	bLedJog : BOOL;
	bLedDistance : BOOL;
	bLedReset : BOOL;
	bLedAlt : BOOL;
	 
	bLedUp : BOOL;
	bLedDown : BOOL;
	bLedLeft : BOOL;
	bLedRight : BOOL;
END_STRUCT
END_TYPE

// ---- POUs/HMI/Provider/HwHmi/Structures/HMI_PROVIDER_HW_IN.TcDUT
TYPE HMI_PROVIDER_HW_IN EXTENDS ST_HMI_IN :
STRUCT
	// HW specific IN
	stP10A_Pult	AT%I* : ST_P10A_Pult_IN;
	
	stP50A_Haupt AT%I* : ST_P50A_Haupt_IN;
	
	stP51A_S1HandBs	AT%I* : ST_P51A_EuchnerHandB_IN;

END_STRUCT
END_TYPE

// ---- POUs/HMI/Provider/HwHmi/Structures/HMI_PROVIDER_HW_OUT.TcDUT
TYPE HMI_PROVIDER_HW_OUT EXTENDS ST_HMI_OUT :
STRUCT
	// HW specific OUT
	stP10A_Pult	AT%Q* : ST_P10A_Pult_OUT;
	
	stP50A_Haupt AT%Q* : ST_P50A_Haupt_OUT;
	
	stP51A_S1HandBs	AT%Q* : ST_P51A_EuchnerHandB_OUT;
	
END_STRUCT
END_TYPE

// ---- POUs/HMI/Provider/HwHmi/Structures/HMI_PROVIDER_HW_IO.TcDUT
TYPE HMI_PROVIDER_HW_IO :
STRUCT
	stIn	: HMI_PROVIDER_HW_IN;
	stOut	: HMI_PROVIDER_HW_OUT;
END_STRUCT
END_TYPE

// ---- POUs/HMI/Provider/HwHmi/Structures/_Base/ST_PxAB_SxHandAsBs_IN.TcDUT
TYPE ST_PxAB_SxHandAsBs_IN :
STRUCT
	//bEs			: BOOL; // Handbediengerät Sx AS/BS - ES
	//bConfirm		: BOOL; // Zustimmung
	//bS4			: BOOL; // res
	//bS5			: BOOL; // res
	bAngleP			: BOOL; // Winkelverstellung Auf; Taste 6
	//bS7			: BOOL; // res
	//bS8			: BOOL; // res
	bAngleN			: BOOL; // Winkelverstellung Ab; Taste 9
	bStpZust01		: BOOL; // Zustellung Schrittweite 0,1mm; Taste 10
	bStpZust001		: BOOL; // Zustellung Schrittweite 0,01mm; Taste 11
	bStpZust0001	: BOOL; // Zustellung Schrittweite 0,001mm; Taste 12
	bZustP			: BOOL; // Zustellung +; Taste 13
	bTravL			: BOOL; // Traversierung links; Taste 14
	
	bResetError		: BOOL; // reset error
	
	bTravR			: BOOL; // Traversierung rechts; Taste 16
	bZustN			: BOOL; // Zustellung -; Taste 17
END_STRUCT
END_TYPE

// ---- POUs/HMI/Provider/HwHmi/Structures/_Base/ST_PxAB_SxHandAsBs_OUT.TcDUT
TYPE ST_PxAB_SxHandAsBs_OUT :
STRUCT
	bLedS4	: BOOL; // LED zu Taste Sx
	bLedS5	: BOOL;
	bLedS6	: BOOL;
	bLedS7	: BOOL;
	bLedS8	: BOOL;
	bLedS9	: BOOL;
	bLedS10	: BOOL;
	bLedS11	: BOOL;
	bLedS12	: BOOL;
	bLedS13	: BOOL;
	bLedS14	: BOOL;
	bLedS15	: BOOL;
	bLedS16	: BOOL;
	bLedS17	: BOOL;
END_STRUCT
END_TYPE

// ---- POUs/HMI/Provider/Tc3Hmi/Structures/Stations/ST_StationToTc3Hmi.TcDUT
TYPE ST_StationToTc3Hmi :
STRUCT
	stStationName			: ST_Text;	//example -> station 001
	
	//astButton				: ARRAY[0..CONST.iMaxIdxLocalButton] OF ST_HMI_BUTTON_OUT; //programmer defined buttons
	
	//stCounter				: ARRAY[0..CONST.iMaxIdxCounter] OF ST_Counter_Item_String;
	//stEingabeStatusColor	: ST_HMI_COLOR_STRING;
	//stEingabeStatus			: ST_Text;
	
END_STRUCT
END_TYPE

// ---- POUs/HMI/Provider/Tc3Hmi/Structures/Stations/ST_StationFromTc3Hmi.TcDUT
TYPE ST_StationFromTc3Hmi :
STRUCT
	astButton						: ARRAY[0..iMaxIdxLocalButton] OF ST_HMI_BUTTON_IN; // station specific buttons
END_STRUCT
END_TYPE

// ---- POUs/HMI/Provider/Tc3Hmi/Structures/ST_FromTc3Hmi.TcDUT
TYPE ST_FromTc3Hmi EXTENDS ST_HMI_IN :
STRUCT
	// general
	eLanguage					: E_Language := E_Language.DE;
	sCurrentPage				: WSTRING;
	sSetTargetPageConfirm		: WSTRING;
	stPopup						: ST_PopUp_FromHmi;
	//stButton_CloseHmi			: ST_Button_FromHmi; //button close hmi
	stControlCounter			: ST_CounterControlIn;	
	
	// stations custom
	//astStation					: ARRAY[0..E_Station.eStation_nMaxIdx] OF ST_StationFromTc3Hmi;
END_STRUCT
END_TYPE

// ---- POUs/HMI/Provider/Tc3Hmi/Structures/ST_Header.TcDUT
TYPE ST_Header :
STRUCT
	stButtonNavUser		: ST_HMI_BUTTON_OUT;
	stMessageBox1		: ST_Text;
	stMessageBox1Color	: ST_HMI_COLOR_STRING;
	stMessageBox2		: ST_Text;
	stMessageBox2Color	: ST_HMI_COLOR_STRING;
	stMessageBox3		: ST_Text;
	stMessageBox3Color	: ST_HMI_COLOR_STRING;
	stStationName		: ST_Text;
	sDateAndTime		: STRING;
	nLanguageList		: INT; //count of laguages
	aLanguageList		: ARRAY[0..5] OF ST_Text;
END_STRUCT
END_TYPE

// ---- POUs/HMI/Provider/Tc3Hmi/Structures/ST_HMI_Tc3.TcDUT
TYPE ST_HMI_Tc3 :
STRUCT
	stIn	: ST_FromTc3Hmi;
	stOut	: ST_ToTc3Hmi;
END_STRUCT
END_TYPE

// ---- POUs/HMI/Provider/Tc3Hmi/Structures/ST_ToTc3Hmi.TcDUT
TYPE ST_ToTc3Hmi EXTENDS ST_HMI_OUT:
STRUCT
	sSetTargetPage				: WSTRING := "Pages/Stations/conStationOverview.content";
	stHeader					: ST_Header;
	
	stPopup						: ST_PopUp_ToHmi;
	
	stCounter					: ARRAY[0..CONST.iMaxIdxCounter] OF ST_Counter_Item_String;
	stControlCounter			: ST_CounterControlOut;
	
	stConditionMonitoring		: ST_ToTc3HmiConditionMonitoring;
	stSetupPlant				: ARRAY[0..30] OF ST_SetupPlant_Item_String;
	stEmergencyStop				: ARRAY[0..20] OF ST_ToTc3Hmi_EmergencyStop;
	stDoor						: ARRAY[0..20] OF ST_ToTc3Hmi_Door;
	
	//stations
	//astStation					: ARRAY[0..E_Station.eStation_nMaxIdx] OF ST_StationToTc3Hmi;
END_STRUCT
END_TYPE

// ---- POUs/HMI/Provider/Tc3Hmi/Structures/ST_ToTc3HmiConditionMonitoring.TcDUT
TYPE ST_ToTc3HmiConditionMonitoring :
STRUCT
	fVoltage_L1	:REAL;
	fVoltage_L2	:REAL;
	fVoltage_L3	:REAL;
	fVoltage_L1_L2 :REAL;
	fVoltage_L2_L3 :REAL;
	fVoltage_L3_L1 :REAL;
	fPowerFactor :REAL;
	fCurrent_L1 :REAL;
	fCurrent_L2 :REAL;
	fCurrent_L3 :REAL;
	fRealPower_L1 :REAL;	//Wirkleistung
	fRealPower_L2 :REAL;	//Wirkleistung
	fRealPower_L3 :REAL;	//Wirkleistung
	fIdlePower_L1 :REAL;	//Blindleistung
	fIdlePower_L2 :REAL;	//Blindleistung
	fIdlePower_L3 :REAL;	//Blindleistung
	fApparentPower_L1 :REAL;	//Scheinleistung
	fApparentPower_L2 :REAL;	//Scheinleistung
	fArrarentPower_L3 :REAL;	//Scheinleistung
END_STRUCT
END_TYPE

// ---- POUs/HMI/Provider/Tc3Hmi/Structures/ST_ToTc3Hmi_Door.TcDUT
TYPE ST_ToTc3Hmi_Door :
STRUCT
	stName			: ST_Text;
	stItem			: ST_Text;
	stStateColor	: ST_HMI_COLOR_STRING;
END_STRUCT
END_TYPE

// ---- POUs/HMI/Provider/Tc3Hmi/Structures/ST_ToTc3Hmi_EmergencyStop.TcDUT
TYPE ST_ToTc3Hmi_EmergencyStop :
STRUCT
	stName			: ST_Text;
	stItem			: ST_Text;
	nState			: INT;	
END_STRUCT
END_TYPE

// ---- POUs/HMI/Provider/Tc3Hmi/Structures/UserControls/DataGrid/ST_UserControlGrid_FromHmi.TcDUT
TYPE ST_UserControlGrid_FromHmi :
STRUCT
	stButtonSave	: ST_HMI_BUTTON_IN;
END_STRUCT
END_TYPE

// ---- POUs/HMI/Provider/Tc3Hmi/Structures/UserControls/DataGrid/ST_UserControlGrid_ToHmi.TcDUT
TYPE ST_UserControlGrid_ToHmi :
STRUCT
	stButtonSave	: ST_HMI_BUTTON_OUT;
END_STRUCT
END_TYPE

// ---- POUs/HMI/Provider/Tc3Hmi/Structures/UserControls/ManualControl Axis/ST_UserControl_Manual_Axis_FromHmi.TcDUT
TYPE ST_UserControl_Manual_Axis_FromHmi :
STRUCT
	fTargetPosition				: REAL;
	eJogMode					: E_Axis_JogMode;
	stButtonJogPos,
	stButtonJogNeg,
	stButtonGoTo,
	stButtonGear,
	stButtonBrake,			
	stButtonSetPos,	
	stButtonRefReset			: ST_HMI_BUTTON_IN;
	nSelectedRowIndex			: UINT;
	nSelectedColumnIndex		: UINT;		
	bTargetListClick			: BOOL;
	bSetTargetClick				: BOOL;
END_STRUCT
END_TYPE

// ---- POUs/HMI/Provider/Tc3Hmi/Structures/UserControls/ManualControl Axis/ST_UserControl_Manual_Axis_Item.TcDUT
TYPE ST_UserControl_Manual_Axis_Item :
STRUCT
	stName	: ST_Text;
	fPos	: LREAL;
END_STRUCT
END_TYPE

// ---- POUs/HMI/Provider/Tc3Hmi/Structures/UserControls/ManualControl Axis/ST_UserControl_Manual_Axis_Item_String.TcDUT
TYPE ST_UserControl_Manual_Axis_Item_String :
STRUCT
	stName				: ST_Text;
	stPos				: ST_Text;
END_STRUCT
END_TYPE

// ---- POUs/HMI/Provider/Tc3Hmi/Structures/UserControls/ManualControl Axis/ST_UserControl_Manual_Axis_ToHmi.TcDUT
TYPE ST_UserControl_Manual_Axis_ToHmi :
STRUCT
	bVisible					: BOOL;
	bVisibleGear				: BOOL;
	bVisibleRefReset			: BOOL;
	bVisibleBrake				: BOOL;
	bVisibleSetPos				: BOOL;
	stObjectName,
	stGearStatus				: ST_Text;
	sOverride					: STRING;
	sTargetPosition				: STRING;
	sActPosition				: STRING;
	stButtonJogPos,
	stButtonJogNeg,
	stButtonGoTo,
	stButtonGear,				
	stButtonBrake,
	stButtonSetPos,
	stButtonRefReset			: ST_HMI_BUTTON_OUT;	
	aJogModeName				: ARRAY[0..5] OF ST_Text;
	stRefStatus					: ST_Text;	
	stTargetList				: ARRAY[1..10] OF ST_UserControl_Manual_Axis_Item_String; /// product data
END_STRUCT
END_TYPE

// ---- POUs/HMI/Provider/Tc3Hmi/Structures/UserControls/ManualControl Cylinder/ST_UserControl_Manual_Cylinder_FromHmi.TcDUT
TYPE ST_UserControl_Manual_Cylinder_FromHmi :
STRUCT
	stButton_Hp,
	stButton_Mp,
	stButton_Wp	: ST_HMI_BUTTON_IN;
END_STRUCT
END_TYPE

// ---- POUs/HMI/Provider/Tc3Hmi/Structures/UserControls/ManualControl Cylinder/ST_UserControl_Manual_Cylinder_ToHmi.TcDUT
TYPE ST_UserControl_Manual_Cylinder_ToHmi :
STRUCT
	bVisible : BOOL;
	stObjectName				: ST_Text;
	stButton_Hp,
	stButton_Mp,
	stButton_Wp	: ST_HMI_BUTTON_OUT;
	bVisible_Button_Mp			: bool;
END_STRUCT
END_TYPE

// ---- POUs/HMI/Provider/Tc3Hmi/Structures/UserControls/ManualControl Device/ST_UserControl_Manual_Device_FromHmi.TcDUT
TYPE ST_UserControl_Manual_Device_FromHmi :
STRUCT
	stOn,
	stOff		: ST_HMI_BUTTON_IN;	
END_STRUCT
END_TYPE

// ---- POUs/HMI/Provider/Tc3Hmi/Structures/UserControls/ManualControl Device/ST_UserControl_Manual_Device_ToHmi.TcDUT
TYPE ST_UserControl_Manual_Device_ToHmi :
STRUCT
	bVisible 		: BOOL;
	stObjectName	: ST_Text;
	stState			: ST_Text;
	stOn,
	stOff			: ST_HMI_BUTTON_OUT;	
END_STRUCT
END_TYPE

// ---- POUs/HMI/Provider/Tc3Hmi/Structures/UserControls/ManualControl Drive/ST_UserControl_Manual_Drive_FromHmi.TcDUT
TYPE ST_UserControl_Manual_Drive_FromHmi :
STRUCT
	eJogMode					: E_Drive_JogMode;
	stButton_Tipp_Pos,
	stButton_Tipp_Neg,
	stButton_Stop				: ST_HMI_BUTTON_IN;
END_STRUCT
END_TYPE

// ---- POUs/HMI/Provider/Tc3Hmi/Structures/UserControls/ManualControl Drive/ST_UserControl_Manual_Drive_ToHmi.TcDUT
TYPE ST_UserControl_Manual_Drive_ToHmi :
STRUCT
	bVisible : BOOL;
	stObjectName				: ST_Text;
	stState						: ST_Text;
	stButton_Tipp_Pos,
	stButton_Tipp_Neg,
	stButton_Stop				: ST_HMI_BUTTON_OUT;
	aDriveModeName				: ARRAY[0..1] OF ST_Text;
END_STRUCT
END_TYPE

// ---- POUs/HMI/Provider/Tc3Hmi/Structures/UserControls/SensorActor/ST_ToVisuSensorActor.TcDUT
TYPE ST_ToVisuSensorActor :
STRUCT
	stType			: ST_Text;
	stName			: ST_Text;
	stBMK			: ST_Text;
	stZustand		: ST_Text;
END_STRUCT
END_TYPE

// ---- POUs/HMI/Provider/_Enumerations/E_HMI_CONTROL_REQUEST.TcDUT
{attribute 'qualified_only'}
{attribute 'strict'}
TYPE E_HMI_CONTROL_REQUEST :
(
	Default,
	RecipeMgmtRequest,
	SettingMgmtRequest,
	UserMgmtRequest
);   	
END_TYPE

// ---- POUs/HMI/Provider/_Enumerations/E_HMI_PROVIDER.TcDUT
{attribute 'qualified_only'}
{attribute 'strict'}
TYPE E_HMI_PROVIDER :
(
	eHmiProvider_none,
	eHmiProvider_HW,
	eHmiProvider_TC3HMI,
	
	// keep this last:
	eHmiProvider_nMaxIdx
);
END_TYPE

// ---- POUs/HMI/_Enumerations/E_Axis_JogMode.TcTLEO
{attribute 'qualified_only'}
{attribute 'strict'}
TYPE E_Axis_JogMode :
(
	eJogMode_0 := 0,//Kontinuierliche Bewegung
	//eJogMode_1, 	//Tippweg
	eJogMode_1,		//0,01 Tippen
	eJogMode_2,		//0,1 Tippen
	eJogMode_3,		//1 Tippen
	eJogMode_4,		//10 Tippen
	eJogMode_5		//100 Tippen
);
END_TYPE

// ---- POUs/HMI/_Enumerations/E_DataType.TcTLEO
{attribute 'qualified_only'}
{attribute 'strict'}
TYPE E_DataType :
(
	eDataType_None := 0,
	eDataType_bool,
	eDataType_int,
	eDataType_lreal,
	eDataType_wstring,
	eDataType_time_ms,
	eDataType_time_s,
	eDataType_time_m,
	eDataType_time_h,
	
	eDataType_Max
);
END_TYPE

// ---- POUs/HMI/_Enumerations/E_Drive_JogMode.TcDUT
{attribute 'qualified_only'}
{attribute 'strict'}
TYPE E_Drive_JogMode :
(
	eJogMode_0 := 0,//Kontinuierliche Bewegung
	eJogMode_1 		//Tipp Bewegung
);
END_TYPE

// ---- POUs/HMI/_Enumerations/E_Language.TcDUT
//{attribute 'qualified_only'}
//{attribute 'strict'}
TYPE E_Language :
(
	// english
	EN := 0,
	// german
	DE,
	// bulgarisch
	BG,
	
	/// zero based max language index
	eLanguage_maxIdx
);
END_TYPE

// ---- POUs/HMI/_Enumerations/E_ManualObjectControlMode.TcDUT
TYPE E_ManualObjectControlMode :
(
	eManualObjectControlMode_none := 0,
	eManualObjectControlMode_cylinder := 1,
	eManualObjectControlMode_device := 2,
	eManualObjectControlMode_servo := 3
);
END_TYPE

// ---- POUs/HMI/_Enumerations/E_Popup.TcDUT
{attribute 'qualified_only'}
{attribute 'strict'}
TYPE E_Popup :
(
	ePopupNone := 0,
	ePopupSafetyEs,
	ePopupStempelkissenWechseln,
	ePopup02,
	ePopup03,
	ePopup04,
	ePopupMax
);
END_TYPE

// ---- POUs/HMI/_Enumerations/E_RecipeMode.TcTLEO
//{attribute 'qualified_only'}
//{attribute 'strict'}
TYPE E_RecipeMode :
(
	eRecipeMode_None := 0,
	eRecipeMode_ToFrom,
	
	eRecipeMode_Max
);
END_TYPE

// ---- POUs/HMI/_Enumerations/E_User.TcTLEO
//{attribute 'qualified_only'}
//{attribute 'strict'}
TYPE E_User :
(
	eUser_none := 0,	(*User | none*)
	eUser_1,			(*User | 1*)
	eUser_2,			(*User | 2*)
	eUser_3,			(*User | 3*)
	eUser_4,			(*User | 4*)
	eUser_5,			(*User | 5*)
	eUser_6,			(*User | 6*)
	eUser_7,			(*User | 7*)
	eUser_8,			(*User | 8*)
	eUser_9,			(*User | 9*)
	eUser_10,			(*User | 10*)

	eUser_11,			(*User | 11*)
	eUser_12,			(*User | 12*)
	eUser_13,			(*User | 13*)
	eUser_14,			(*User | 14*)
	eUser_15,			(*User | 15*)
	eUser_16,			(*User | 16*)
	eUser_17,			(*User | 17*)
	eUser_18,			(*User | 18*)
	eUser_19,			(*User | 19*)
	eUser_20,			(*User | 20*)	
(*Maximum*)
	eUser_nMaxIdx
);
END_TYPE

// ---- POUs/HMI/_Enumerations/E_User_Level.TcDUT
//{attribute 'qualified_only'}
//{attribute 'strict'}
{attribute 'to_string'}
{attribute 'to_wstring'}
TYPE E_User_Level :
(
	eUser_Level_none := 0,			(*user level 0 = none 1= Operator 2 = Plant Manager 3 = maintenance 4 = reserve 5= admin*)
	eUser_Level_Operator,			(* 1 = Bediener*)
	eUser_Level_Manager,			(* 2 = Einsteller*)
	eUser_Level_Maintenance,		(* 3 = Instandhalter*)
	eUser_Level_Level4,				(* 4 = Reserve*)
	eUser_Level_Admin,				(* 5 = Administrator *)
	eUser_Level_Programmer,			(* 6 = Programmer *)

(*Maximum*)
	eUser_Level_nMaxIdx
);
END_TYPE

// ---- POUs/HMI/_Structures/Counter/E_CounterReaction.TcTLEO
//{attribute 'qualified_only'}
//{attribute 'strict'}
TYPE E_CounterReaction :
(
	eCounterReaction_None := 0,
	eCounterReaction_Info,
	eCounterReaction_Warning,
	eCounterReaction_Error,
	eCounterReaction_SerialFault_Warning,
	eCounterReaction_SerialFault_Error,
	
	eCounterReaction_Max
);
END_TYPE

// ---- POUs/HMI/_Structures/Counter/ST_CounterControlIn.TcDUT
TYPE ST_CounterControlIn :
STRUCT
	stButtonSave		: ST_HMI_BUTTON_IN;
	stButtonReset		: ST_HMI_BUTTON_IN;	
	nSelectedRowIndex	: UINT;
	nSelectedColumIndex	: UINT;
	nInputBool			: DINT;
	nInputNumber		: DINT;
	wsInputString		: WSTRING;
	eUserLevel			: E_User_Level;	
	eReaction			: E_CounterReaction;	
END_STRUCT
END_TYPE

// ---- POUs/HMI/_Structures/Counter/ST_CounterControlOut.TcDUT
TYPE ST_CounterControlOut :
STRUCT
	stButtonSave		: ST_HMI_BUTTON_OUT;
	stButtonReset		: ST_HMI_BUTTON_OUT;		
	bVisible_UserLevel	: BOOL;
	nUserLevelUsers		: INT; //count of recipe mode list
	aUserLevelUsers		: ARRAY[0..E_User_Level.eUser_Level_nMaxIdx] OF ST_Text;
	bVisible_Reaction	: BOOL;
	nReaction			: INT; //count of recipe mode list
	aReaction			: ARRAY[0..E_CounterReaction.eCounterReaction_Max] OF ST_Text;	
	bVisible_Number		: BOOL;
	bVisible_String		: BOOL;
	bVisibleInfo		: BOOL;
	stInfo				: ST_Text;
END_STRUCT
END_TYPE

// ---- POUs/HMI/_Structures/Counter/ST_Counter_Item_String.TcDUT
TYPE ST_Counter_Item_String :
STRUCT
	stIndex					:ST_Text;
	stGroup					:ST_Text;
	stName					:ST_Text;
	stValueOk				:ST_Text;	
	stValueNok				:ST_Text;
	stValueTotal			:ST_Text;	
	stValueOkLevel1			:ST_Text;
	stReactionOkLevel1		:ST_Text;
	stValueOkLevel2			:ST_Text;
	stReactionOkLevel2		:ST_Text;
	stValueNokLevel1		:ST_Text;
	stReactionNokLevel1		:ST_Text;
	stValueNokLevel2		:ST_Text;
	stReactionNokLevel2		:ST_Text;
	stValueTotalLevel1		:ST_Text;
	stReactionTotalLevel1	:ST_Text;
	stValueTotalLevel2		:ST_Text;
	stReactionTotalLevel2	:ST_Text;		
	stUserLevel				:ST_Text;
	stDataType				:ST_Text;	
END_STRUCT
END_TYPE

// ---- POUs/HMI/_Structures/Data/ST_Data_Item_String.TcDUT
TYPE ST_Data_Item_String :
STRUCT
	stIndex				:ST_Text;
	stGroup				:ST_Text;
	stName				:ST_Text;
	stValue				:ST_Text;
	stValueMin			:ST_Text;
	stValueMax			:ST_Text;	
	stUnit				:ST_Text;
	stUserLevel			:ST_Text;
	stDataType			:ST_Text;
	stRecipeMode		:ST_Text;
END_STRUCT
END_TYPE

// ---- POUs/HMI/_Structures/Monitoring/ST_GridObject_Name_Value1_Event1_Value2_Event2_Unit.TcDUT
TYPE ST_GridObject_Name_Value1_Event1_Value2_Event2_Unit :
STRUCT
	sGroup				:STRING;
	sName				:STRING;
	fValue1				:LREAL;
	fValue1Min			:LREAL;
	fValue1Max			:LREAL;
	iEvent1				:INT;	//exampe : no reaction=0 reaction 1..x = 1..x
	fValue2				:LREAL;
	fValue2Min			:LREAL;
	fValue2Max			:LREAL;
	iEvent2				:INT;	//exampe : no reaction=0 reaction 1..x = 1..x
	bYesNo				:BOOL;
	sUnit				:STRING;
END_STRUCT
END_TYPE

// ---- POUs/HMI/_Structures/Monitoring/ST_GridObject_Name_sValue_Unit.TcDUT
TYPE ST_GridObject_Name_sValue_Unit :
STRUCT
	sGroup				:STRING;
	sName				:STRING;
	sValue				:STRING;
	sValueMin			:STRING;
	sValueMax			:STRING;
	bYesNo				:BOOL;
	sUnit				:STRING;
END_STRUCT
END_TYPE

// ---- POUs/HMI/_Structures/Monitoring/ST_Monitoring_Station.TcDUT
TYPE ST_Monitoring_Station EXTENDS ST_Monitoring_Base :
STRUCT
	astMonitoring		: ARRAY[0..CONST.iMaxIdxMonitoring] OF ST_Data_Item;
	astMonitoringView	: ARRAY[0..CONST.iMaxIdxMonitoring] OF ST_Data_Item_String;
END_STRUCT
END_TYPE

// ---- POUs/HMI/_Structures/Monitoring/ST_Monitoring.TcDUT
TYPE ST_Monitoring :
STRUCT
	astMonitoringGlobal		: ARRAY[0..CONST.iMaxIdxMonitoring] OF ST_Data_Item;				// general/global monitoring
	astMonitoringModule		: ARRAY[0..E_Module.eModule_nMaxIdx] OF ST_Monitoring_Module;		// module monitoring
	astMonitoringStation	: ARRAY[0..E_Station.eStation_nMaxIdx] OF ST_Monitoring_Station;	// station monitoring
END_STRUCT
END_TYPE

// ---- POUs/HMI/_Structures/Data/ST_Data_Item.TcDUT
TYPE ST_Data_Item :
STRUCT
	stIndex		: ST_Text;
	stGroup		: ST_Text;
	stName		: ST_Text;
	
	bValue		: BOOL;
	tValue		: TIME;
	sValue		: WSTRING;
	nValue		: INT;
	fValue		: LREAL;
	fValueMin	: LREAL;
	fValueMax	: LREAL;
	
	stUnit		: ST_Text;
	eUserLevel	: E_User_Level;
	eDataType	: E_DataType;
	eRecipeMode	: E_RecipeMode;
END_STRUCT
END_TYPE

// ---- POUs/HMI/_Structures/Monitoring/ST_Monitoring_Base.TcDUT
TYPE ST_Monitoring_Base :
STRUCT
	sGroup				: STRING;
	stName				: ST_Text;
	bManual				: BOOL;
	bInHome				: BOOL;
	bAuto				: BOOL;;
	bBusy				: BOOL;
	bWarning			: BOOL;
	bError				: BOOL;
	bTransferEnable		: BOOL;
END_STRUCT
END_TYPE

// ---- POUs/HMI/_Structures/Monitoring/ST_Monitoring_Module.TcDUT
TYPE ST_Monitoring_Module EXTENDS ST_Monitoring_Base :
STRUCT
	astMonitoring		: ARRAY[0..CONST.iMaxIdxMonitoring] OF ST_Data_Item;
	astMonitoringView	: ARRAY[0..CONST.iMaxIdxMonitoring] OF ST_Data_Item_String;
END_STRUCT
END_TYPE

// ---- POUs/HMI/_Structures/Popup/E_PopupSymbol.TcDUT
{attribute 'qualified_only'}
{attribute 'strict'}
TYPE E_PopupSymbol :
(
	ePopupSymbolNone := 0,
	ePopupSymbolOk,
	ePopupSymbolNok
);
END_TYPE

// ---- POUs/HMI/_Structures/Popup/ST_PopUp_FromHmi.TcDUT
TYPE ST_PopUp_FromHmi :
STRUCT
	stButton01	: ST_HMI_BUTTON_IN;
	stButton02	: ST_HMI_BUTTON_IN;
	stButton03	: ST_HMI_BUTTON_IN;
	stButton04	: ST_HMI_BUTTON_IN;
END_STRUCT
END_TYPE

// ---- POUs/HMI/_Structures/Popup/ST_PopUp_ToHmi.TcDUT
TYPE ST_PopUp_ToHmi :
STRUCT
	bVisible		: BOOL;
	nSymbol			: INT; //E_PopupSymbol;
	stText			: ST_Text;
	bButton01		: BOOL := TRUE;
	stButton01		: ST_HMI_BUTTON_OUT;
	bButton02		: BOOL := TRUE;
	stButton02		: ST_HMI_BUTTON_OUT;
	bButton03		: BOOL := TRUE;
	stButton03		: ST_HMI_BUTTON_OUT;
	bButton04		: BOOL := TRUE;
	stButton04		: ST_HMI_BUTTON_OUT;
END_STRUCT
END_TYPE

// ---- POUs/HMI/_Structures/Recipe/ST_HMI_RECIPE_IN.TcDUT
TYPE ST_HMI_RECIPE_IN :
STRUCT
	// Current Recipe Infos
	bSaveCurrentRecipe				:BOOL;
	
	
	// Recipe Management
	
	wsNewEditRecipeName				:WSTRING(255); // Read/Write
	wsNewEditRecipeComment			:WSTRING(255); // Read/Write
	wsNewEditRecipeProduct			:WSTRING(255); // Read/Write
	bCreateNewRecipe				:BOOL;
	bUpdateRecipe					:BOOL;
	
	nSelectedRecipe					:INT;
	bRefreshRecipeList				:BOOL;
	bLoadSelectedRecipe				:BOOL;
	bDeleteSelectedRecipe			:BOOL;
	wsCopyRecipeNewName				:WSTRING(255); // Read/Write
	bCopySelectedRecipe				:BOOL;
	
END_STRUCT
END_TYPE

// ---- POUs/HMI/_Structures/Recipe/ST_HMI_RECIPE_OUT.TcDUT
TYPE ST_HMI_RECIPE_OUT :
STRUCT
	// Current Recipe Infos
	
	wsActiveRecipe					: WSTRING(255); // Read/Write
	wsActiveRecipeComment			: WSTRING(255); // Read/Write
	wsActiveRecipeProduct			: WSTRING(255); // Read/Write
	wsActiveRecipeSavedInfo			: WSTRING(80);
	bEnableSaveCurrentRecipe		: BOOL;
	                                  
	                                  
	// Recipe Management              
	bEnableCreateNewRecipe			: BOOL;
	bEnableUpdateRecipe				: BOOL;
                                      
	aRecipeList						: ARRAY[0..iMaxIdxRecipe] OF WSTRING(255);
	nMaxEntryRecipeList				: INT;
	bEnableLoadRecipe				: BOOL;
	bEnableDeleteRecipe				: BOOL;
	bEnableCopyRecipe				: BOOL;
                                      
	stStatusText					: ST_Text;
	stStatusColor					: ST_HMI_COLOR_STRING;
	bStatusTextVisible				: BOOL;
END_STRUCT
END_TYPE

// ---- POUs/HMI/_Structures/Safety/ST_HMI_SAFETY_IN.TcDUT
TYPE ST_HMI_SAFETY_IN :
STRUCT
	bQuitSafety,
	
	bQuitAreaST10,
	bUnlockDoorST33	: BOOL;
END_STRUCT
END_TYPE

// ---- POUs/HMI/_Structures/Safety/ST_HMI_SAFETY_OUT.TcDUT
TYPE ST_HMI_SAFETY_OUT :
STRUCT
	// Safety Infos
	
	/// EmergencyStop/Not-Halt Status von Safety (TRUE = OK)
	bSAFE_ES_Ok				: BOOL;
	
	/// State of every emergency stop button (TRUE = OK)
	bSAFE_EStop_State		: ARRAY[0..E_EmergencyStop.eEmergencyStop_nMaxIdx] OF BOOL;
	
	/// Schutzbereich OK von Safety (TRUE = OK)
	bSAFE_AREA_Ok			: ARRAY[0..iSafety_Anzahl_Schutzbereiche] OF BOOL;
	bSAFE_AREA_Ok_Color		: ARRAY[0..iSafety_Anzahl_Schutzbereiche] OF ST_HMI_COLOR_STRING;
	
	/// GATE OK von Safety (TRUE = OK)
	stSAFE_GATE_Ok_Color	: ARRAY[0..E_Door.eDoor_nMaxIdx] OF ST_HMI_COLOR_STRING;
			
	/// Zustimmeinrichtung von Safety (TRUE = OK)
	bSAFE_CONFIRMDEVICE_OK	: BOOL;
	
	bLedResetSafety,
	bLedResetAreaST10,
	bLedResetAreaST33		: BOOL;
END_STRUCT
END_TYPE

// ---- POUs/HMI/_Structures/Settngs/ST_HMI_CONTROL_SETTING_IN.TcDUT
TYPE ST_HMI_CONTROL_SETTING_IN :
STRUCT
	stControlSetting_Plant		: ST_HMI_CONTROL_SETTING_ITEM_IN;
	stControlSetting_Product	: ST_HMI_CONTROL_SETTING_ITEM_IN;
	stControlSetting_Production	: ST_HMI_CONTROL_SETTING_ITEM_IN;	
	
	astControlSetting_Modules	: ARRAY[0..E_Module.eModule_nMaxIdx] OF ST_HMI_CONTROL_SETTING_ITEM_IN;
	astControlSetting_Stations	: ARRAY[0..E_Station.eStation_nMaxIdx] OF ST_HMI_CONTROL_SETTING_ITEM_IN;
END_STRUCT
END_TYPE

// ---- POUs/HMI/_Structures/Settngs/ST_HMI_CONTROL_SETTING_OUT.TcDUT
TYPE ST_HMI_CONTROL_SETTING_OUT :
STRUCT
	stControlSetting_Plant		: ST_HMI_CONTROL_SETTING_ITEM_OUT;
	stControlSetting_Product	: ST_HMI_CONTROL_SETTING_ITEM_OUT;
	stControlSetting_Production	: ST_HMI_CONTROL_SETTING_ITEM_OUT;

	stSettingViewPlant			: ARRAY[0..E_PlantSettings.ePlantSetting_nMaxIdx] OF ST_Data_Item_String;
	stSettingViewProduct		: ARRAY[0..E_ProductSettings.eProductSettings_nMaxIdx] OF ST_Data_Item_String;
	stSettingViewProduction		: ARRAY[0..E_ProductionSettings.eProductionSettings_nMaxIdx] OF ST_Data_Item_String;	

	astSettingModules			: ARRAY[0..E_Module.eModule_nMaxIdx] OF ST_HMI_CONTROL_SETTING_MODULE_OUT;
	astSettingStations			: ARRAY[0..E_Station.eStation_nMaxIdx] OF ST_HMI_CONTROL_SETTING_STATION_OUT;
END_STRUCT
END_TYPE

// ---- POUs/HMI/_Structures/Settngs/ST_HMI_CONTROL_SETTING_STATION_OUT.TcDUT
TYPE ST_HMI_CONTROL_SETTING_STATION_OUT :
STRUCT
	stControlSetting	: ST_HMI_CONTROL_SETTING_ITEM_OUT;
	stSettingView		: ARRAY[0..CONST.iMaxIdxLocalSetting] OF ST_Data_Item_String;
END_STRUCT
END_TYPE

// ---- POUs/HMI/_Structures/Settngs/ST_HMI_CONTROL_SETTING_MODULE_OUT.TcDUT
TYPE ST_HMI_CONTROL_SETTING_MODULE_OUT :
STRUCT
	stControlSetting	: ST_HMI_CONTROL_SETTING_ITEM_OUT;
	stSettingView		: ARRAY[0..CONST.iMaxIdxLocalSetting] OF ST_Data_Item_String;
END_STRUCT
END_TYPE

// ---- POUs/HMI/_Structures/SetupPlant/E_SetupPlantShape.TcDUT
TYPE E_SetupPlantShape :
(
	eSetupPlantShape_None := 0,
	eSetupPlantShape_DreieckGruen,
	eSetupPlantShape_DreieckRot,
	
	eSetupPlantShape_ViereckViolett := 11,
	eSetupPlantShape_ViereckRosa,
	
	eSetupPlantShape_SechseckBlau := 21,
	eSetupPlantShape_SechseckGelb,	
	
	eSetupPlantShape_KreisGruen := 31,
	eSetupPlantShape_KreisRosa,	
	
	eSetupPlantShape_Max
);
END_TYPE

// ---- POUs/HMI/_Structures/SetupPlant/E_SetupPlantStateShape.TcDUT
TYPE E_SetupPlantStateShape :
(
	eSetupPlantStateShape_None := 0,
	eSetupPlantStateShape_Nok,
	eSetupPlantStateShape_Ok,
	
	
	eSetupPlantStateShape_Max
);
END_TYPE

// ---- POUs/HMI/_Structures/SetupPlant/ST_SetupPlant_Item_String.TcDUT
TYPE ST_SetupPlant_Item_String :
STRUCT
	stGroup					:ST_Text;	
	stStation				:ST_Text;
	stName					:ST_Text;
	stSet					:ST_Text;
	stGet					:ST_Text;	
	stState					:ST_Text;		
	stUserLevel				:ST_Text;
	stDataType				:ST_Text;	
END_STRUCT
END_TYPE

// ---- POUs/HMI/_Structures/Settngs/ST_HMI_CONTROL_SETTING_ITEM_IN.TcDUT
TYPE ST_HMI_CONTROL_SETTING_ITEM_IN :
STRUCT
	stButtonSave		: ST_HMI_BUTTON_IN;
	nSelectedRowIndex	: UINT;
	nSelectedColumIndex	: UINT;
	bInputBool			: BOOL;
	nInputNumber		: INT;
	fInputFloat			: REAL;
	wsInputString		: WSTRING;
	eUserLevel			: E_User_Level;
	eRecipeMode			: E_RecipeMode;
END_STRUCT
END_TYPE

// ---- POUs/HMI/_Structures/Settngs/ST_HMI_CONTROL_SETTING_ITEM_OUT.TcDUT
TYPE ST_HMI_CONTROL_SETTING_ITEM_OUT :
STRUCT
	stButtonSave		: ST_HMI_BUTTON_OUT;
	bVisible_RecipeMode	: BOOL;
	nRecipeMode			: INT; //count of recipe mode list
	aRecipeMode			: ARRAY[0..E_RecipeMode.eRecipeMode_Max] OF ST_Text;
	
	bVisible_UserLevel	: BOOL;
	bVisible_Bool		: BOOL;
	bVisible_Float		: BOOL;
	bVisible_Number		: BOOL;
	bVisible_String		: BOOL;
	bVisibleInfo		: BOOL;
	stInfo				: ST_Text;
	
	nUserLevelUsers		: INT; //count of recipe mode list
	aUserLevelUsers		: ARRAY[0..E_User_Level.eUser_Level_nMaxIdx] OF ST_Text;
END_STRUCT
END_TYPE

// ---- POUs/HMI/_Structures/ST_HMI.TcDUT
TYPE ST_HMI :
STRUCT
	stIn 	: ST_HMI_IN;
	stOut 	: ST_HMI_OUT;
END_STRUCT
END_TYPE

// ---- POUs/HMI/_Structures/ST_HMI_IN.TcDUT
TYPE ST_HMI_IN EXTENDS ST_HMI_BASE_IN :
STRUCT
	// additional, project specific stuff:
	iOverride		: INT;
	
	stM001 	: ST_M001_HMI_IN;
	stSt010 : ST_St010_HMI_IN;
	stSt020 : ST_St020_HMI_IN;
	stSt030 : ST_St030_HMI_IN;
	stSt040 : ST_St040_HMI_IN;
END_STRUCT
END_TYPE

// ---- POUs/HMI/_Structures/ST_HMI_InOut.TcDUT
TYPE ST_HMI_InOut :
STRUCT
	/// HMI direct (IN/OUT) struct
	/// e.g. for accessing (r/w) project specific settings

	//stM001 	: ST_M001_HMI_InOut;
	
	stSt010		: ST_St010_HMI_IN_OUT;
	stSt020		: ST_St020_HMI_IN_OUT;
	stSt030		: ST_St030_HMI_IN_OUT;
	stSt040		: ST_St040_HMI_IN_OUT;
	
	// global axis manager
	stHmiAxisManager	: ST_HmiAxisManager;
END_STRUCT
END_TYPE

// ---- POUs/HMI/_Structures/ST_HMI_OUT.TcDUT
TYPE ST_HMI_OUT : //EXTENDS ST_HMI_BASE_OUT :
STRUCT
	// note, ST_HMI_BASE_OUT is not inherited anymoredue to performance issues in provider mapping
	stCommon			: REFERENCE TO ST_HMI_BASE_OUT;
	
	// additional, project specific stuff:
	stButtonDoorOpen	: ST_HMI_BUTTON_OUT;
	stButtonDoorClose	: ST_HMI_BUTTON_OUT;
	stButtonConfirm		: ST_HMI_BUTTON_OUT;
	
	stM001 : ST_M001_HMI_OUT;
	stSt010 : ST_St010_HMI_OUT;
	stSt020 : ST_St020_HMI_OUT;
	stSt030 : ST_St030_HMI_OUT;
	stSt040 : ST_St040_HMI_OUT;
END_STRUCT
END_TYPE

// ---- POUs/HMI/_Structures/ST_NameValue.TcDUT
TYPE ST_NameValue :
STRUCT
	sName 	: STRING(31);
	sValue 	: STRING; 
END_STRUCT
END_TYPE

// ---- POUs/HMI/_Structures/UserManagment/ST_HMI_USER_MGMT_IN.TcDUT
TYPE ST_HMI_USER_MGMT_IN :
STRUCT
	stControlObject					: ST_HMI_GRID_IN;
	sUserManagment_InputString		: STRING;	//Input String Values
	sUserManagment_InputPassword	: STRING;	//Input Password Login
	nUserManagment_InputNumeric		: INT;		//Input Numeric Values
	nUserManagment_InputUserLevel	: INT;		//Input DropDown UserLevel
	stButton_LogOut					: ST_HMI_BUTTON_IN;		//Logout Button
	stButton_LogIn					: ST_HMI_BUTTON_IN;		//Login Button
	stButton_Submit					: ST_HMI_BUTTON_IN;		//Übernehmen Button

	bDeleteUser						: BOOL;
	sCreateDeleteUserName			: STRING;
	sCreateDeleteUserNameConfirm	: STRING;
	sCreateUser_InputPassword		: STRING;	//Input Password Login for create new user
	
	// for Beckhoff HMI UserMgmt:
	iHmiUserLevel					: INT;
END_STRUCT
END_TYPE

// ---- POUs/HMI/_Structures/UserManagment/ST_HMI_USER_MGMT_OUT.TcDUT
TYPE ST_HMI_USER_MGMT_OUT :
STRUCT
	sUserState						: STRING;
	stButton_LogOut					: ST_HMI_BUTTON_OUT;
	stButton_LogIn					: ST_HMI_BUTTON_OUT;
	stButton_Submit					: ST_HMI_BUTTON_OUT;
	stUserLevel						: ARRAY [0..20] OF ST_User_Management;
	bUserLevel						: ARRAY [0..E_User_Level.eUser_Level_nMaxIdx] OF BOOL;
	aUserLevelList					: ARRAY[0..E_User_Level.eUser_Level_nMaxIdx] OF ST_Text;
	bKeyboardInputVisible			: BOOL;
	bNumpadInputVisible				: BOOL;
	bUserLevelInputVisible			: BOOL;
	bPasswordInputVisible			: BOOL;
	stUserManagementMessage			: ST_Text;
	
	stInputDisplayText				: ST_Text;

	bCreateDeleteUserVisible		: BOOL;
	stInfo							: ST_Text;
END_STRUCT
END_TYPE

// ---- POUs/HMI/_Structures/UserManagment/ST_User_Management.TcDUT
{attribute 'pack_mode' := '1'}
TYPE ST_User_Management :
STRUCT
	sName 				: STRING;
	sPassword			: STRING;
	iUserLevel			: E_User_Level;
	stUserLevelName		: ST_Text;
	iUserLevelMin		: INT;
	iUserLevelMax		: INT;
END_STRUCT
END_TYPE

// ---- POUs/HMI/_Structures/_Base/Button/ST_HMI_BUTTON_IN.TcDUT
TYPE ST_HMI_BUTTON_IN :
STRUCT
	bClick	: BOOL;
END_STRUCT
END_TYPE

// ---- POUs/HMI/_Structures/_Base/Button/ST_HMI_BUTTON_OUT.TcDUT
TYPE ST_HMI_BUTTON_OUT :
STRUCT
	stName	: ST_Text;				// button text (e.g. for SW button)
	stColor	: ST_HMI_COLOR_STRING;	// button color (e.g. for SW button)
	bLed	: BOOL;					// LED (e.g. for HW button)
END_STRUCT
END_TYPE

// ---- POUs/HMI/_Structures/_Base/Common/ST_HMI_BASE_CONTROL_IN.TcDUT
TYPE ST_HMI_BASE_CONTROL_IN :
STRUCT
	// control
	stButton_Start,
	stButton_CycleStop,
	stButton_Stop,
	stButton_Home,
	stButton_Step,
	stButton_Reset 		: ST_HMI_BUTTON_IN;
	
	// OP modes
	stButton_OPM_Auto,
	stButton_OPM_Step,
	stButton_OPM_Manual	: ST_HMI_BUTTON_IN;
	
END_STRUCT
END_TYPE

// ---- POUs/HMI/_Structures/_Base/Common/ST_HMI_BASE_CONTROL_OUT.TcDUT
TYPE ST_HMI_BASE_CONTROL_OUT :
STRUCT
	// control
	stButton_Home 			: ST_HMI_BUTTON_OUT;
	stButton_Step			: ST_HMI_BUTTON_OUT;
	stButton_Reset			: ST_HMI_BUTTON_OUT;
	stButton_CycleStop		: ST_HMI_BUTTON_OUT;
	stButton_Start			: ST_HMI_BUTTON_OUT;
	stButton_Stop			: ST_HMI_BUTTON_OUT;
	stButton_PlantLight		: ST_HMI_BUTTON_OUT;
	                                              
	// OP modes
	stButton_OPM_Auto,
	stButton_OPM_Step,
	stButton_OPM_Manual		: ST_HMI_BUTTON_OUT;
	
	// info
	stSwitch_OPM_1,
	stSwitch_OPM_2,
	stSwitch_OPM_3,
	stSwitch_OPM_4,
	stInfo1,
	stInfo2					: ST_Text;

	stColorSwitch_OPM_1,
	stColorSwitch_OPM_2,
	stColorSwitch_OPM_3,
	stColorSwitch_OPM_4		: ST_HMI_COLOR_STRING;			
END_STRUCT
END_TYPE

// ---- POUs/HMI/_Structures/_Base/Common/ST_HMI_BASE_SPECIAL_IN.TcDUT
TYPE ST_HMI_BASE_SPECIAL_IN:
STRUCT
	stButton_LedTest				: ST_HMI_BUTTON_IN;
	stButton_CloseHmi				: ST_HMI_BUTTON_IN;
	stButton_SetSystemTime			: ST_HMI_BUTTON_IN;
	stButton_Eplan					: ST_HMI_BUTTON_IN;
	stButton_Calculator				: ST_HMI_BUTTON_IN;
	stButton_KeyenceAutoIdNetwNav	: ST_HMI_BUTTON_IN;
	stButton_KeyenceIv2Nav			: ST_HMI_BUTTON_IN;
	stButton_CleanScreen			: ST_HMI_BUTTON_IN;
END_STRUCT
END_TYPE

// ---- POUs/HMI/_Structures/_Base/Common/ST_HMI_GRID_IN.TcDUT
TYPE ST_HMI_GRID_IN :
STRUCT
	nSelectedRowIndex	: UINT;
	nSelectedColumIndex	: UINT;	
END_STRUCT
END_TYPE

// ---- POUs/HMI/_Structures/_Base/Common/ST_HMI_NAME_VALUE_STRING.TcDUT
TYPE ST_HMI_NAME_VALUE_STRING :
STRUCT
	stName	: ST_Text;
	stPos	: ST_Text;
END_STRUCT
END_TYPE

// ---- POUs/HMI/_Structures/_Base/Common/ST_HMI_TRAFFIC_LIGHT_OUT.TcDUT
TYPE ST_HMI_TRAFFIC_LIGHT_OUT :
STRUCT
	bLedGN	: BOOL;
	bLedGE	: BOOL;
	bLedRT	: BOOL;
	bLedBL	: BOOL;
END_STRUCT
END_TYPE

// ---- POUs/HMI/_Structures/_Base/Manual/ManualControl Axis/ST_HMI_MANUAL_AXIS_IN.TcDUT
TYPE ST_HMI_MANUAL_AXIS_IN :
STRUCT
	fTargetPosition		: REAL;
	eJogMode			: E_Axis_JogMode;
	
	stButtonJogPos,
	stButtonJogNeg,
	stButtonGoTo,
	stButtonGear,
	stButtonBrake,			
	stButtonSetPos,	// ToDo: chk nicht verwendet?
	stButtonRefReset	: ST_HMI_BUTTON_IN;
	
	nSelectedRowIndex	: UINT;
	bSetTargetFromList	: BOOL;
	bSetTarget			: BOOL;
END_STRUCT
END_TYPE

// ---- POUs/HMI/_Structures/_Base/Manual/ManualControl Axis/ST_HMI_MANUAL_AXIS_ITEM.TcDUT
TYPE ST_HMI_MANUAL_AXIS_ITEM :
STRUCT
	stName	: ST_Text;
	fPos	: REAL;
END_STRUCT
END_TYPE

// ---- POUs/HMI/_Structures/_Base/Manual/ManualControl Axis/ST_HMI_MANUAL_AXIS_ITEM_STRING.TcDUT
TYPE ST_HMI_MANUAL_AXIS_ITEM_STRING :
STRUCT
	stName	: ST_Text;
	stPos	: ST_Text;
END_STRUCT
END_TYPE

// ---- POUs/HMI/_Structures/_Base/Manual/ManualControl Axis/ST_HMI_MANUAL_AXIS_OUT.TcDUT
TYPE ST_HMI_MANUAL_AXIS_OUT :
STRUCT
	bVisible			: BOOL;
	bVisibleGear		: BOOL;
	bVisibleRefReset	: BOOL;
	bVisibleBrake		: BOOL;
	bVisibleSetPos		: BOOL;
	stObjectName,
	stGearStatus		: ST_Text;
	sOverride			: STRING;
	sTargetPosition		: STRING;
	sActPosition		: STRING;
	stButtonJogPos,
	stButtonJogNeg,
	stButtonGoTo,
	stButtonGear,				
	stButtonBrake,
	stButtonSetPos,
	stButtonRefReset	: ST_HMI_BUTTON_OUT;
	aJogModeName		: ARRAY[0..5] OF ST_Text;
	stRefStatus			: ST_Text;	
	stTargetList		: ARRAY[0..9] OF ST_HMI_NAME_VALUE_STRING;
END_STRUCT
END_TYPE

// ---- POUs/HMI/_Structures/_Base/Manual/ManualControl Cylinder/ST_HMI_MANUAL_CYLINDER_IN.TcDUT
TYPE ST_HMI_MANUAL_CYLINDER_IN :
STRUCT	
	stButtonHp,
	stButtonMp,
	stButtonWp	: ST_HMI_BUTTON_IN;
END_STRUCT
END_TYPE

// ---- POUs/HMI/_Structures/_Base/Manual/ManualControl Cylinder/ST_HMI_MANUAL_CYLINDER_OUT.TcDUT
TYPE ST_HMI_MANUAL_CYLINDER_OUT :
STRUCT
	bVisible		: BOOL;
	stObjectName	: ST_Text;
	stButtonHp,
	stButtonMp,
	stButtonWp		: ST_HMI_BUTTON_OUT;
	bMpVisible		: BOOL;
END_STRUCT
END_TYPE

// ---- POUs/HMI/_Structures/_Base/Manual/ManualControl Device/ST_HMI_MANUAL_DEVICE_IN.TcDUT
TYPE ST_HMI_MANUAL_DEVICE_IN :
STRUCT
	stButtonOn,
	stButtonOff	: ST_HMI_BUTTON_IN;
	
	fValue		: REAL;
END_STRUCT
END_TYPE

// ---- POUs/HMI/_Structures/_Base/Manual/ManualControl Device/ST_HMI_MANUAL_DEVICE_OUT.TcDUT
TYPE ST_HMI_MANUAL_DEVICE_OUT :
STRUCT
	bVisible,
	bValueVisible	: BOOL;
	stObjectName,
	stState,
	stValueText		: ST_Text;
	stButtonOn,
	stButtonOff		: ST_HMI_BUTTON_OUT;	
END_STRUCT
END_TYPE

// ---- POUs/HMI/_Structures/_Base/Manual/ManualControl Drive/ST_HMI_MANUAL_DRIVE_IN.TcDUT
TYPE ST_HMI_MANUAL_DRIVE_IN :
STRUCT
	eJogMode		: E_Drive_JogMode;
	stButtonJogPos,
	stButtonJogNeg,
	stButtonStop	: ST_HMI_BUTTON_IN;
END_STRUCT
END_TYPE

// ---- POUs/HMI/_Structures/_Base/Manual/ManualControl Drive/ST_HMI_MANUAL_DRIVE_OUT.TcDUT
TYPE ST_HMI_MANUAL_DRIVE_OUT :
STRUCT
	bVisible			: BOOL;
	stObjectName		: ST_Text;
	stState				: ST_Text;
	stButtonJogPos,
	stButtonJogNeg,
	stButtonStop		: ST_HMI_BUTTON_OUT;
	aDriveModeName		: ARRAY[0..1] OF ST_Text;
END_STRUCT
END_TYPE

// ---- POUs/HMI/_Structures/_Base/Module/ST_HMI_BASE_MODULE_IN.TcDUT
TYPE ST_HMI_BASE_MODULE_IN EXTENDS ST_HMI_BASE_CONTROL_IN:
STRUCT
	stButtonNavigation	: ST_HMI_BUTTON_IN;
	iStepchain			: INT; //ToDo: iStepchain HMI -> PLC STATION!?!?! (mapping missing)
	stManual			: ST_HMI_BASE_MODULE_MANUAL_IN;
END_STRUCT
END_TYPE

// ---- POUs/HMI/_Structures/_Base/Module/ST_HMI_BASE_MODULE_MANUAL_IN.TcDUT
TYPE ST_HMI_BASE_MODULE_MANUAL_IN :
STRUCT
	diSelectedObjectIndex	: DINT;
	stManualCylinder		: ST_HMI_MANUAL_CYLINDER_IN;
	stManualDrive			: ST_HMI_MANUAL_DRIVE_IN;
	stManualAxis			: ST_HMI_MANUAL_AXIS_IN;
	stManualDevice			: ST_HMI_MANUAL_DEVICE_IN;	
END_STRUCT
END_TYPE

// ---- POUs/HMI/_Structures/_Base/Module/ST_HMI_BASE_MODULE_MANUAL_OUT.TcDUT
TYPE ST_HMI_BASE_MODULE_MANUAL_OUT :
STRUCT
	bManualMode			: BOOL;	
	stManualCylinder	: ST_HMI_MANUAL_CYLINDER_OUT;
	stManualDrive		: ST_HMI_MANUAL_DRIVE_OUT;
	stManualAxis		: ST_HMI_MANUAL_AXIS_OUT;
	stManualDevice		: ST_HMI_MANUAL_DEVICE_OUT;
	
	stObjects			: ARRAY[0..iMaxIdxObject] OF ST_Object_Item; // e.g.: fbAxis, ...	
END_STRUCT
END_TYPE

// ---- POUs/HMI/_Structures/_Base/Module/ST_HMI_BASE_MODULE_OUT.TcDUT
TYPE ST_HMI_BASE_MODULE_OUT EXTENDS ST_HMI_BASE_CONTROL_OUT :
STRUCT
	stName				: ST_Text;
	stButtonNavigation	: ST_HMI_BUTTON_OUT;
	
	// info
	stState_Auto,
	stState_Home,
	stState				: ST_Text;	
	nStepChainName		: INT; // count visible rows from array aStepChainName
	aStepChainName		: ARRAY[0..CONST.iMaxIdxLocalStepChain] OF ST_Text;
	
	stManual			: ST_HMI_BASE_MODULE_MANUAL_OUT;
END_STRUCT
END_TYPE

// ---- POUs/HMI/_Structures/_Base/Station/ST_HMI_BASE_STATION_IN.TcDUT
TYPE ST_HMI_BASE_STATION_IN EXTENDS ST_HMI_BASE_CONTROL_IN:
STRUCT
	stButtonNavigation	: ST_HMI_BUTTON_IN;
	iStepchain			: INT; //ToDo: iStepchain HMI -> PLC STATION!?!?! (mapping missing)
	stManual			: ST_HMI_BASE_STATION_MANUAL_IN;
END_STRUCT
END_TYPE

// ---- POUs/HMI/_Structures/_Base/Station/ST_HMI_BASE_STATION_MANUAL_IN.TcDUT
TYPE ST_HMI_BASE_STATION_MANUAL_IN :
STRUCT
	diSelectedObjectIndex	: DINT;
	stControl				: ST_HMI_GRID_IN;
	stManualCylinder		: ST_HMI_MANUAL_CYLINDER_IN;
	stManualDrive			: ST_HMI_MANUAL_DRIVE_IN;
	stManualAxis			: ST_HMI_MANUAL_AXIS_IN;
	stManualDevice			: ST_HMI_MANUAL_DEVICE_IN;	
END_STRUCT
END_TYPE

// ---- POUs/HMI/_Structures/_Base/Station/ST_HMI_BASE_STATION_MANUAL_OUT.TcDUT
TYPE ST_HMI_BASE_STATION_MANUAL_OUT :
STRUCT
	bManualMode			: BOOL;	
	stManualCylinder	: ST_HMI_MANUAL_CYLINDER_OUT;
	stManualDrive		: ST_HMI_MANUAL_DRIVE_OUT;
	stManualAxis		: ST_HMI_MANUAL_AXIS_OUT;
	stManualDevice		: ST_HMI_MANUAL_DEVICE_OUT;
	
	stObjects			: ARRAY[0..iMaxIdxObject] OF ST_Object_Item; // e.g.: fbAxis, ...	
END_STRUCT
END_TYPE

// ---- POUs/HMI/_Structures/_Base/Station/ST_HMI_BASE_STATION_OUT.TcDUT
TYPE ST_HMI_BASE_STATION_OUT EXTENDS ST_HMI_BASE_CONTROL_OUT :
STRUCT
	stName				: ST_Text;
	stButtonNavigation	: ST_HMI_BUTTON_OUT;
	
	// info
	stState_Auto,
	stState_Home,
	stState_Station		: ST_Text;	
	nStepChainName		: INT; // count visible rows from array aStepChainName
	aStepChainName		: ARRAY[0..CONST.iMaxIdxLocalStepChain] OF ST_Text;
	
	stManual			: ST_HMI_BASE_STATION_MANUAL_OUT;
END_STRUCT
END_TYPE

// ---- POUs/HMI/_Structures/_Base/ST_HMI_BASE_IN.TcDUT
TYPE ST_HMI_BASE_IN :
STRUCT
	stMain 			: ST_HMI_BASE_CONTROL_IN;
	arrStModule		: ARRAY[0..E_Module.eModule_nMaxIdx] OF ST_HMI_BASE_Module_IN;
	arrStStation	: ARRAY[0..E_Station.eStation_nMaxIdx] OF ST_HMI_BASE_STATION_IN;
	
	stRecipe 		: ST_HMI_RECIPE_IN;
	stSettings 		: ST_HMI_CONTROL_SETTING_IN;
	stSafety		: ST_HMI_SAFETY_IN;
	stSpecial		: ST_HMI_BASE_SPECIAL_IN;
	stUserMgmt		: ST_HMI_USER_MGMT_IN;
END_STRUCT
END_TYPE

// ---- POUs/HMI/_Structures/_Base/ST_HMI_BASE_OUT.TcDUT
TYPE ST_HMI_BASE_OUT :
STRUCT
	stMain			: ST_HMI_BASE_CONTROL_OUT;
	arrStModule		: ARRAY[0..E_Module.eModule_nMaxIdx] OF ST_HMI_BASE_Module_OUT;
	arrStStation	: ARRAY[0..E_Station.eStation_nMaxIdx] OF ST_HMI_BASE_STATION_OUT;
	
	stRecipe		: ST_HMI_RECIPE_OUT; 	// Recipe Management structure
	stSettings 		: ST_HMI_CONTROL_SETTING_OUT;
	stMonitoring	: ST_Monitoring;		// monitoring to hmi or data bench
	stSafety		: ST_HMI_SAFETY_OUT;	// Safety info
	stUserMgmt		: ST_HMI_USER_MGMT_OUT;
	stTrafficLight	: ST_HMI_TRAFFIC_LIGHT_OUT;
	
	aSystemInfos	: ARRAY[0..CONST.iMaxIdxSystemInfo] OF ST_NameValue;
END_STRUCT
END_TYPE

// ---- POUs/HMI/_Structures/_Common/ST_HexColor.TcDUT
{attribute 'pack_mode' := '1'}
TYPE  ST_HexColor:
STRUCT
	
	(*	Color Hexcode...[generiert aus .net]		*)
	ActiveBorder :DINT:=16#D4D0C8;
	ActiveCaption :DINT:=16#0054E3;
	ActiveCaptionText :DINT:=16#FFFFFF;
	AliceBlue :DINT:=16#F0F8FF;
	AntiqueWhite :DINT:=16#FAEBD7;
	AppWorkspace :DINT:=16#808080;
	Aqua :DINT:=16#00FFFF;
	Aquamarine :DINT:=16#7FFFD4;
	Azure :DINT:=16#F0FFFF;
	Beige :DINT:=16#F5F5DC;
	Bisque :DINT:=16#FFE4C4;
	Black :DINT:=16#000000;
	BlanchedAlmond :DINT:=16#FFEBCD;
	Blue :DINT:=16#0000FF;
	BlueViolet :DINT:=16#8A2BE2;
	Brown :DINT:=16#A52A2A;
	BurlyWood :DINT:=16#DEB887;
	ButtonFace :DINT:=16#ECE9D8;
	ButtonHighlight :DINT:=16#FFFFFF;
	ButtonShadow :DINT:=16#ACA899;
	CadetBlue :DINT:=16#5F9EA0;
	Chartreuse :DINT:=16#7FFF00;
	Chocolate :DINT:=16#D2691E;
	Control :DINT:=16#ECE9D8;
	ControlDark :DINT:=16#ACA899;
	ControlDarkDark :DINT:=16#716F64;
	ControlLight :DINT:=16#F1EFE2;
	ControlLightLight :DINT:=16#FFFFFF;
	ControlText :DINT:=16#000000;
	Coral :DINT:=16#FF7F50;
	CornflowerBlue :DINT:=16#6495ED;
	Cornsilk :DINT:=16#FFF8DC;
	Crimson :DINT:=16#DC143C;
	Cyan :DINT:=16#00FFFF;
	DarkBlue :DINT:=16#00008B;
	DarkCyan :DINT:=16#008B8B;
	DarkGoldenrod :DINT:=16#B8860B;
	DarkGray :DINT:=16#A9A9A9;
	DarkGreen :DINT:=16#006400;
	DarkKhaki :DINT:=16#BDB76B;
	DarkMagenta :DINT:=16#8B008B;
	DarkOliveGreen :DINT:=16#556B2F;
	DarkOrange :DINT:=16#FF8C00;
	DarkOrchid :DINT:=16#9932CC;
	DarkRed :DINT:=16#8B0000;
	DarkSalmon :DINT:=16#E9967A;
	DarkSeaGreen :DINT:=16#8FBC8B;
	DarkSlateBlue :DINT:=16#483D8B;
	DarkSlateGray :DINT:=16#2F4F4F;
	DarkTurquoise :DINT:=16#00CED1;
	DarkViolet :DINT:=16#9400D3;
	DeepPink :DINT:=16#FF1493;
	DeepSkyBlue :DINT:=16#00BFFF;
	Desktop :DINT:=16#004E98;
	DimGray :DINT:=16#696969;
	DodgerBlue :DINT:=16#1E90FF;
	Firebrick :DINT:=16#B22222;
	FloralWhite :DINT:=16#FFFAF0;
	ForestGreen :DINT:=16#228B22;
	Fuchsia :DINT:=16#FF00FF;
	Gainsboro :DINT:=16#DCDCDC;
	GhostWhite :DINT:=16#F8F8FF;
	Gold :DINT:=16#FFD700;
	Goldenrod :DINT:=16#DAA520;
	GradientActiveCaption :DINT:=16#3D95FF;
	GradientInactiveCaption :DINT:=16#9DB9EB;
	Gray :DINT:=16#808080;
	GrayText :DINT:=16#ACA899;
	Green :DINT:=16#008000;
	GreenYellow :DINT:=16#ADFF2F;
	Highlight :DINT:=16#316AC5;
	HighlightText :DINT:=16#FFFFFF;
	Honeydew :DINT:=16#F0FFF0;
	HotPink :DINT:=16#FF69B4;
	HotTrack :DINT:=16#000080;
	InactiveBorder :DINT:=16#D4D0C8;
	InactiveCaption :DINT:=16#7A96DF;
	InactiveCaptionText :DINT:=16#D8E4F8;
	IndianRed :DINT:=16#CD5C5C;
	Indigo :DINT:=16#4B0082;
	Info :DINT:=16#FFFFE1;
	InfoText :DINT:=16#000000;
	Ivory :DINT:=16#FFFFF0;
	Khaki :DINT:=16#F0E68C;
	Lavender :DINT:=16#E6E6FA;
	LavenderBlush :DINT:=16#FFF0F5;
	LawnGreen :DINT:=16#7CFC00;
	LemonChiffon :DINT:=16#FFFACD;
	LightBlue :DINT:=16#ADD8E6;
	LightCoral :DINT:=16#F08080;
	LightCyan :DINT:=16#E0FFFF;
	LightGoldenrodYellow :DINT:=16#FAFAD2;
	LightGray :DINT:=16#D3D3D3;
	LightGreen :DINT:=16#90EE90;
	LightPink :DINT:=16#FFB6C1;
	LightSalmon :DINT:=16#FFA07A;
	LightSeaGreen :DINT:=16#20B2AA;
	LightSkyBlue :DINT:=16#87CEFA;
	LightSlateGray :DINT:=16#778899;
	LightSteelBlue :DINT:=16#B0C4DE;
	LightYellow :DINT:=16#FFFFE0;
	Lime :DINT:=16#00FF00;
	LimeGreen :DINT:=16#32CD32;
	Linen :DINT:=16#FAF0E6;
	Magenta :DINT:=16#FF00FF;
	Maroon :DINT:=16#800000;
	MediumAquamarine :DINT:=16#66CDAA;
	MediumBlue :DINT:=16#0000CD;
	MediumOrchid :DINT:=16#BA55D3;
	MediumPurple :DINT:=16#9370DB;
	MediumSeaGreen :DINT:=16#3CB371;
	MediumSlateBlue :DINT:=16#7B68EE;
	MediumSpringGreen :DINT:=16#00FA9A;
	MediumTurquoise :DINT:=16#48D1CC;
	MediumVioletRed :DINT:=16#C71585;
	Menu :DINT:=16#FFFFFF;
	MenuBar :DINT:=16#ECE9D8;
	MenuHighlight :DINT:=16#316AC5;
	MenuText :DINT:=16#000000;
	MidnightBlue :DINT:=16#191970;
	MintCream :DINT:=16#F5FFFA;
	MistyRose :DINT:=16#FFE4E1;
	Moccasin :DINT:=16#FFE4B5;
	NavajoWhite :DINT:=16#FFDEAD;
	Navy :DINT:=16#000080;
	OldLace :DINT:=16#FDF5E6;
	Olive :DINT:=16#808000;
	OliveDrab :DINT:=16#6B8E23;
	Orange :DINT:=16#FFA500;
	OrangeRed :DINT:=16#FF4500;
	Orchid :DINT:=16#DA70D6;
	PaleGoldenrod :DINT:=16#EEE8AA;
	PaleGreen :DINT:=16#98FB98;
	PaleTurquoise :DINT:=16#AFEEEE;
	PaleVioletRed :DINT:=16#DB7093;
	PapayaWhip :DINT:=16#FFEFD5;
	PeachPuff :DINT:=16#FFDAB9;
	Peru :DINT:=16#CD853F;
	Pink :DINT:=16#FFC0CB;
	Plum :DINT:=16#DDA0DD;
	PowderBlue :DINT:=16#B0E0E6;
	Purple :DINT:=16#800080;
	Red :DINT:=16#FF0000;
	RosyBrown :DINT:=16#BC8F8F;
	RoyalBlue :DINT:=16#4169E1;
	SaddleBrown :DINT:=16#8B4513;
	Salmon :DINT:=16#FA8072;
	SandyBrown :DINT:=16#F4A460;
	ScrollBar :DINT:=16#D4D0C8;
	SeaGreen :DINT:=16#2E8B57;
	SeaShell :DINT:=16#FFF5EE;
	Sienna :DINT:=16#A0522D;
	Silver :DINT:=16#C0C0C0;
	SkyBlue :DINT:=16#87CEEB;
	SlateBlue :DINT:=16#6A5ACD;
	SlateGray :DINT:=16#708090;
	Snow :DINT:=16#FFFAFA;
	SpringGreen :DINT:=16#00FF7F;
	SteelBlue :DINT:=16#4682B4;
	TTAN :DINT:=16#D2B48C;
	Teal :DINT:=16#008080;
	Thistle :DINT:=16#D8BFD8;
	Tomato :DINT:=16#FF6347;
	//Transparent :DINT:=16#FFFFFF;
	Turquoise :DINT:=16#40E0D0;
	Violet :DINT:=16#EE82EE;
	Wheat :DINT:=16#F5DEB3;
	White :DINT:=16#FFFFFF;
	WhiteSmoke :DINT:=16#F5F5F5;
	Window :DINT:=16#FFFFFF;
	WindowFrame :DINT:=16#000000;
	WindowText :DINT:=16#000000;
	Yellow :DINT:=16#FFFF00;
	YellowGreen :DINT:=16#9ACD32;
	GrassGreen	: DINT := 16#ADE204;
END_STRUCT
END_TYPE

// ---- POUs/HMI/_Structures/_Common/ST_HMI_COLOR_STRING.TcDUT
TYPE ST_HMI_COLOR_STRING : STRUCT
	color: STRING; (* Defining a color as CSS color: #hexadecimal, rgb(), rgba(), hsl(), hsla(), css color keyword, none or transparent. *)
END_STRUCT
END_TYPE

// ---- POUs/HMI/_Structures/_Common/ST_Text.TcDUT
TYPE ST_Text :
STRUCT
	nNameId		: INT;		//example simatic hmi
	wsNameId	: WSTRING; 	//beckhoff tc3 hmi
	wsName		: WSTRING;	//standard name only english
END_STRUCT
END_TYPE

// ---- POUs/HMI/_Structures/_TextLists/ST_Text_List_Components.TcDUT
TYPE ST_Text_List_Components :
STRUCT
	// Mettler Scale
	stText_MettlerACT305_DeviceError	: ST_Text := (
											nNameId:= 1,
											wsNameId:= "Mettler_scale_device_rror",
											wsName:= "Mettler scale device error");	
	stText_MettlerACT305_WatchdError	: ST_Text := (
											nNameId:= 1,
											wsNameId:= "Mettler_scale_watchdog_error",
											wsName:= "Mettler scale watchdog error");	


	// Axis Driver
	stText_AxisUi_PosDirectionWarn		: ST_Text := (
											nNameId:= 1,
											wsNameId:= "Axis_Pos_Dir_Locked",
											wsName:= "Positive Richtung durch Freigabesignal gesperrt");	
	stText_AxisUi_NegDirectionWarn		: ST_Text := (
											nNameId:= 1,
											wsNameId:= "Axis_Neg_Dir_Locked",
											wsName:= "Negative Richtung durch Freigabesignal gesperrt");	
	
	stText_Axis_DriveNotReady			: ST_Text := (
											nNameId:= 1,
											wsNameId:= "Axis_DriveNotReady",
											wsName:= "Antrieb nicht bereit");	
	stText_Axis_SafetyError				: ST_Text := (
											nNameId:= 1,
											wsNameId:= "Axis_SafetyError",
											wsName:= "Safety Fehler -> Reset");	
	stText_Axis_MovingNotReleased		: ST_Text := (
											nNameId:= 1,
											wsNameId:= "Axis_MovingNotReleased",
											wsName:= "Fahrfreigabe nicht vorhanden");	
	stText_Axis_TargetOutOfArea			: ST_Text := (
											nNameId:= 1,
											wsNameId:= "Axis_TargetOutOfArea",
											wsName:= "Zielposition ausserhalb Bereich");	
	stText_Axis_HwNotReady				: ST_Text := (
											nNameId:= 1,
											wsNameId:= "Axis_HwNotReady",
											wsName:= "Antriebshardware nicht bereit");
	stText_Axis_FbError					: ST_Text := (
											nNameId:= 1,
											wsNameId:= "Axis_FbError",
											wsName:= "FB-FehlerNr");
	stText_Axis_NcError					: ST_Text := (
											nNameId:= 1,
											wsNameId:= "Axis_NcError",
											wsName:= "Nc-FehlerNr");
	stText_Axis_HwError					: ST_Text := (
											nNameId:= 1,
											wsNameId:= "Axis_HwError",
											wsName:= "HW-FehlerNr");

	// Sensor
	stText_Sensor_NotOK_True					: ST_Text := (
											nNameId:= 1,
											wsNameId:= "Sensor_NotOKTrue",
											wsName:= "Sensor nicht Belegt");
											
	stText_Sensor_NotOK_False					: ST_Text := (
											nNameId:= 1,
											wsNameId:= "Sensor_NotOKFalse",
											wsName:= "Sensor nicht Frei");											
											
	stText_Sensor_Free					: ST_Text := (
											nNameId:= 1,
											wsNameId:= "Sensor_Free",
											wsName:= "Frei");
	stText_Sensor_Proven				: ST_Text := (
											nNameId:= 1,
											wsNameId:= "Sensor_Proven",
											wsName:= "Belegt");
															
END_STRUCT
END_TYPE

// ---- POUs/HMI/_Structures/_TextLists/ST_Text_List_Global.TcDUT
TYPE ST_Text_List_Global :
STRUCT
	stText_System				: ST_Text_List_System; //System Texte
	stText_Empty				: ST_Text;
	
	//----------------------------------------------------------------------------------------------------
	//language	
	stText_EN				: ST_Text := (
									nNameId:= 1,
									wsNameId:= "l_english",
									wsName:= "English");

	stText_DE				: ST_Text := (
									nNameId:= 1,
									wsNameId:= "l_german",
									wsName:= "Deutsch");

	stText_BE				: ST_Text := (
									nNameId:= 1,
									wsNameId:= "l_belarusisch",
									wsName:= "Belarusisch");	
									
	stText_Null				: ST_Text := (
									nNameId:= 1,
									wsNameId:= "",
									wsName:= "");									
									
	//----------------------------------------------------------------------------------------------------
	//Stepchains
	
	stText_Stepchain01				: ST_Text := (
									nNameId:= 1,
									wsNameId:= "stepchain01",
									wsName:= "step chain 01");
	
	stText_Stepchain02				: ST_Text := (
									nNameId:= 1,
									wsNameId:= "stepchain02",
									wsName:= "step chain 02");
	
	stText_Stepchain03				: ST_Text := (
									nNameId:= 1,
									wsNameId:= "stepchain03",
									wsName:= "step chain 03");
									
	stText_Stepchain04				: ST_Text := (
									nNameId:= 1,
									wsNameId:= "stepchain04",
									wsName:= "step chain 04");
									
	stText_Stepchain05				: ST_Text := (
									nNameId:= 1,
									wsNameId:= "stepchain05",
									wsName:= "step chain 05");
									
	stText_Stepchain06				: ST_Text := (
									nNameId:= 1,
									wsNameId:= "stepchain06",
									wsName:= "step chain 06");
	
	stText_Stepchain07				: ST_Text := (
									nNameId:= 1,
									wsNameId:= "stepchain07",
									wsName:= "step chain 07");
					
	stText_Stepchain08				: ST_Text := (
									nNameId:= 1,
									wsNameId:= "stepchain08",
									wsName:= "step chain 08");
									
	stText_Stepchain09				: ST_Text := (
									nNameId:= 1,
									wsNameId:= "stepchain09",
									wsName:= "step chain 09");
									
	stText_Stepchain10				: ST_Text := (
									nNameId:= 1,
									wsNameId:= "stepchain10",
									wsName:= "step chain 10");
									
	//----------------------------------------------------------------------------------------------------
	//user level
	stText_UserLevel00				: ST_Text := (
									nNameId:= 1,
									wsNameId:= "userlevel00",
									wsName:= "kein Benutzer");
									
	stText_UserLevel01				: ST_Text := (
									nNameId:= 1,
									wsNameId:= "userlevel01",
									wsName:= "Bediener");
									
	stText_UserLevel02				: ST_Text := (
									nNameId:= 1,
									wsNameId:= "userlevel02",
									wsName:= "Einsteller");

	stText_UserLevel03				: ST_Text := (
									nNameId:= 1,
									wsNameId:= "userlevel03",
									wsName:= "Instandhalter");

	stText_UserLevel04				: ST_Text := (
									nNameId:= 1,
									wsNameId:= "userlevel04",
									wsName:= "Reserve");

	stText_UserLevel05				: ST_Text := (
									nNameId:= 1,
									wsNameId:= "userlevel05",
									wsName:= "Administrator");
									
	stText_UserLevel06				: ST_Text := (
									nNameId:= 1,
									wsNameId:= "userlevel06",
									wsName:= "Programmer");	

	//----------------------------------------------------------------------------------------------------
	//counter
	stText_Counter_Reaction_None	: ST_Text := (
									nNameId:= 1,
									wsNameId:= "none",
									wsName:= "keine");

	stText_Counter_Reaction_Info	: ST_Text := (
									nNameId:= 1,
									wsNameId:= "info",
									wsName:= "Info");

	stText_Counter_Reaction_Warning	: ST_Text := (
									nNameId:= 1,
									wsNameId:= "warning",
									wsName:= "Warnung");
									
	stText_Counter_Reaction_Error	: ST_Text := (
									nNameId:= 1,
									wsNameId:= "error",
									wsName:= "Fehler");									

	stText_Counter_Reaction_SerialError_Warning	: ST_Text := (
									nNameId:= 1,
									wsNameId:= "serialerrorwarning",
									wsName:= "Serienfehler Warnung");
									
	stText_Counter_Reaction_SerialError_Warning_Stop	: ST_Text := (
									nNameId:= 1,
									wsNameId:= "serialerrorstop",
									wsName:= "Serienfehler Stop");															
									
	//----------------------------------------------------------------------------------------------------
	//units
	stText_notextempty			: ST_Text := (
									nNameId:= 1,
									wsNameId:= "",
									wsName:= "");	
	
	stText_notext				: ST_Text := (
									nNameId:= 1,
									wsNameId:= "notext",
									wsName:= "notext");	
									
	stText_text					: ST_Text := (
									nNameId:= 1,
									wsNameId:= "text",
									wsName:= "text");	

	stText_name					: ST_Text := (
									nNameId:= 1,
									wsNameId:= "name",
									wsName:= "name");									
	
	stText_percent				: ST_Text := (
									nNameId:= 1,
									wsNameId:= "%",
									wsName:= "%");								
									
	stText_n					: ST_Text := (
									nNameId:= 1,
									wsNameId:= "n",
									wsName:= "n");	

	stText_bool					: ST_Text := (
									nNameId:= 1,
									wsNameId:= "bool",
									wsName:= "bool");
									
	stText_m					: ST_Text := (
									nNameId:= 1,
									wsNameId:= "m",
									wsName:= "m");
	
	stText_mm					: ST_Text := (
									nNameId:= 1,
									wsNameId:= "mm",
									wsName:= "mm");
										
	stText_cm					: ST_Text := (
									nNameId:= 1,
									wsNameId:= "cm",
									wsName:= "cm");
									
	stText_um					: ST_Text := (
									nNameId:= 1,
									wsNameId:= "µm",
									wsName:= "µm");

	stText_Celsius_C			: ST_Text := (
									nNameId:= 1,
									wsNameId:= "C°",
									wsName:= "C°");

	stText_time_ms				: ST_Text := (
									nNameId:= 1,
									wsNameId:= "time_ms",
									wsName:= "ms");
									
	stText_time_s				: ST_Text := (
									nNameId:= 1,
									wsNameId:= "time_s",
									wsName:= "s");

	stText_time_m				: ST_Text := (
									nNameId:= 1,
									wsNameId:= "time_min",
									wsName:= "Min");

	stText_time_h				: ST_Text := (
									nNameId:= 1,
									wsNameId:= "time_hour",
									wsName:= "Std");
									
	stText_time_day				: ST_Text := (
									nNameId:= 1,
									wsNameId:= "time_day",
									wsName:= "day");
									
	stText_time_week				: ST_Text := (
									nNameId:= 1,
									wsNameId:= "time_week",
									wsName:= "week");
									
	stText_time_year				: ST_Text := (
									nNameId:= 1,
									wsNameId:= "time_year",
									wsName:= "year");

	stText_mms						: ST_Text := (
									nNameId:= 1,
									wsNameId:= "velo_mms",
									wsName:= "mm/s");

	stText_mmpmin					: ST_Text := (
									nNameId:= 1,
									wsNameId:= "velo_mm_min",
									wsName:= "mm/min");									
									
	stText_mmin						: ST_Text := (
									nNameId:= 1,
									wsNameId:= "velo_mmin",
									wsName:= "m/min");
									
	stText_mps						: ST_Text := (
									nNameId:= 1,
									wsNameId:= "velo_ms",
									wsName:= "m/s");
									
	stText_degree					: ST_Text := (
									nNameId:= 1,
									wsNameId:= "pos_grad",
									wsName:= "°");
									
	stText_degreeCelsius			: ST_Text := (
									nNameId:= 1,
									wsNameId:= "temp_gradC",
									wsName:= "°C");
									
	stText_degreeS					: ST_Text := (
									nNameId:= 1,
									wsNameId:= "velo_grads",
									wsName:= "°/sec");	
									
	stText_degreeMin				: ST_Text := (
									nNameId:= 1,
									wsNameId:= "velo_gradmin",
									wsName:= "°/min");
									
	stText_gramm					: ST_Text := (
									nNameId:= 1,
									wsNameId:= "gramm",
									wsName:= "g");
									
	stText_kgramm					: ST_Text := (
									nNameId:= 1,
									wsNameId:= "kilogramm",
									wsName:= "kg");
									
	stText_umin						: ST_Text := (
									nNameId:= 1,
									wsNameId:= "roundspermin",
									wsName:= "U/min");
									
	stText_Hz						: ST_Text := (
									nNameId:= 1,
									wsNameId:= "frequncy",
									wsName:= "Hz");
									
	stText_us						: ST_Text := (
									nNameId:= 1,
									wsNameId:= "roundspersec",
									wsName:= "U/s");
									
	stText_Nm						: ST_Text := (
									nNameId:= 1,
									wsNameId:= "Nm",
									wsName:= "Nm");	
	
	stText_Watt						: ST_Text := (
									nNameId:= 1,
									wsNameId:= "Watt",
									wsName:= "W");	
									
	stText_Joule					: ST_Text := (
									nNameId:= 1,
									wsNameId:= "Joule",
									wsName:= "J");	
									
	stText_Drehzahl					: ST_Text := (
									nNameId:= 1,
									wsNameId:= "rotSpeed",
									wsName:= "Drehzahl");
									
	stText_PlantSpeed				: ST_Text := (
									nNameId:= 1,
									wsNameId:= "plantspeed",
									wsName:= "Anlage Geschwindigkeit");	

	stText_PlantSpeedOverride		: ST_Text := (
									nNameId:= 1,
									wsNameId:= "plantspeedoverride",
									wsName:= "Anlage Geschwindigkeit Override");

	stText_Ok						: ST_Text := (
									nNameId:= 1,
									wsNameId:= "ok",
									wsName:= "Io");

	stText_Nok						: ST_Text := (
									nNameId:= 1,
									wsNameId:= "nok",
									wsName:= "Nio");

	stText_Yes						: ST_Text := (
									nNameId:= 1,
									wsNameId:= "yes",
									wsName:= "yes");

	stText_No						: ST_Text := (
									nNameId:= 1,
									wsNameId:= "no",
									wsName:= "no");	

	stText_Tested					: ST_Text := (
									nNameId:= 1,
									wsNameId:= "tested",
									wsName:= "tested");

	stText_NotTested					: ST_Text := (
									nNameId:= 1,
									wsNameId:= "nottested",
									wsName:= "not tested");
									
									
	stText_Settings					: ST_Text := (
									nNameId:= 1,
									wsNameId:= "settings",
									wsName:= "Settings");
									
//----------------------------------------------------------------------------------------------------
//general FBs (EC, ...)

	stText_UnknownError			: ST_Text := (
										wsNameId:= "unknownerror",
										wsName:= "Unbekannter Fehler");

	stText_CheckboundError			: ST_Text := (
										wsNameId:= "checkbounderror",
										wsName:= "Checkbound error");
											
	stText_EcGetSlaveIdentityErr	: ST_Text := (
										wsNameId:= "ecgetslaveidentityerror",
										wsName:= "Fehler bei Slave-Identifizierung");
									
	stText_EcGetSlaveNameErr		: ST_Text := (
										wsNameId:= "ecgetslavenameerror",
										wsName:= "Fehler bei Slave-Namenbestimmung");
									
	stText_EcGetAllSlaveAddrErr		: ST_Text := (
										wsNameId:= "ecgetallslaveaddrerror",
										wsName:= "Fehler bei Slave-Adressbestimmung");
									
	stText_EcCoeSdoReadErr			: ST_Text := (
										wsNameId:= "eccoesdoreaderror",
										wsName:= "Fehler beim Lesen EC COE SDO");
										
	stText_EcCoeHistoryDiag			: ST_Text := (
										wsNameId:= "eccoehistorydiagerror",
										wsName:= "Fehler beim Lesen EC COE Historie");
										
	stText_JobNotSupported			: ST_Text := (
										wsNameId:= "stText_JobNotSupported",
										wsName:= "Job nicht unterstützt");
										
	stText_TimeoutHandshake			: ST_Text := (
										wsNameId:= "stText_TimeoutHandshake",
										wsName:= "Timeout Handshake");
			
	stText_TimeoutCarrier			: ST_Text := (
										wsNameId:= "stText_TimeoutCarrier",
										wsName:= "Timeout WT");
										
	stText_TimeoutCncMachining		: ST_Text := (
										wsNameId:= "stText_TimeoutCncMachining",
										wsName:= "Timeout CNC Bearbeitung");
										
	stText_FixingCylinderNotHP			: ST_Text := (
										wsNameId:= "stText_FixingCylinderNotHP",
										wsName:= "Fixierzylinder nicht in GRST (HP)");
										
	stText_FixingCylinderNotWP			: ST_Text := (
										wsNameId:= "stText_FixingCylinderNotWP",
										wsName:= "Fixierzylinder nicht in AP");
										
	stText_GripperCylinderNotWP		: ST_Text := (
										wsNameId:= "stText_GripperCylinderNotWP",
										wsName:= "Greiferzylinder nicht in AP");
										
	stText_TimeoutReadRFID			: ST_Text := (
										wsNameId:= "stText_TimeoutReadRFID",
										wsName:= "Timeout RFID Lesekopf");
										
	stText_CarrierEmptyRfid			: ST_Text := (
										wsNameId:= "stText_CarrierEmptyRfid",
										wsName:= "WT RFID ist leer");
										
	stText_UnexpectedCarrier		: ST_Text := (
										wsNameId:= "stText_UnexpectedCarrier",
										wsName:= "Unerwarteter WT in Station");
										
	stText_CarrierBufferFull		: ST_Text := (
										wsNameId:= "stText_CarrierBufferFull",
										wsName:= "WT Buffer ist voll");
										
	stText_TrayBufferFull			: ST_Text := (
										wsNameId:= "stText_TrayBufferFull",
										wsName:= "Tray Puffer ist voll");
										
	stText_CarrierNotFound			: ST_Text := (
										wsNameId:= "stText_CarrierNotFound",
										wsName:= "WT nicht gefunden");
										
	stText_CarrierSuspect			: ST_Text := (
										wsNameId:= "stText_CarrierSuspect",
										wsName:= "WT unbekannt");
										
	stText_WrongPartStateNest1		: ST_Text := (
										wsNameId:= "stText_WrongPartStateNest1",
										wsName:= "Ungültiger Teilestatus in Nest 1");
										
	stText_MissingPartNest1			: ST_Text := (
										wsNameId:= "stText_MissingPartNest1",
										wsName:= "Fehlender Teil in Nest 1");
										
	stText_UnexpectedPartNest1		: ST_Text := (
										wsNameId:= "stText_UnexpectedPartNest1",
										wsName:= "Unerwarteter Teil in Nest 1");
										
	stText_WrongPartStateNest2		: ST_Text := (
										wsNameId:= "stText_WrongPartStateNest2",
										wsName:= "Ungültiger Teilestatus in Nest 2");
										
	stText_MissingPartNest2			: ST_Text := (
										wsNameId:= "stText_MissingPartNest2",
										wsName:= "Fehlender Teil in Nest 2");
										
	stText_UnexpectedPartNest2		: ST_Text := (
										wsNameId:= "stText_UnexpectedPartNest2",
										wsName:= "Unerwarteter Teil in Nest 2");
										
	stText_CrashDetection			: ST_Text := (
										wsNameId:= "stText_CrashDetection",
										wsName:= "Crash Sensor ausgelöst");
										
	stText_WrongPartStateRawPartEmco	: ST_Text := (
										wsNameId:= "stText_WrongPartStateRawPartEmco",
										wsName:= "Ungültiger Teilestatus Rohteil in EMCO");

	stText_WrongPartStateFinishPartEmco	: ST_Text := (
										wsNameId:= "stText_WrongPartStateFinishPartEmco",
										wsName:= "Ungültiger Teilestatus Fertigteil in EMCO");
									
//----------------------------------------------------------------------------------------------------
//objects
											
	stText_ObjectTypeAxis			: ST_Text := (
									nNameId:= 1,
									wsNameId:= "objecttypeaxis",
									wsName:= "objecttypeaxis");
									
	stText_ObjectTypeCylinder		: ST_Text := (
									nNameId:= 1,
									wsNameId:= "objecttypecylinder",
									wsName:= "objecttypecylinder");	
									
	stText_ObjectTypeDrive		: ST_Text := (
									nNameId:= 1,
									wsNameId:= "objecttypedrive",
									wsName:= "objecttypedrive");									

	stText_ObjectTypeDevice		: ST_Text := (
									nNameId:= 1,
									wsNameId:= "objecttypedevice",
									wsName:= "objecttypedevice");

	//----------------------------------------------------------------------------------------------------
	//control
	stText_On		: ST_Text := (
									nNameId:= 1,
									wsNameId:= "on",
									wsName:= "on");	
									
	stText_Off		: ST_Text := (
									nNameId:= 1,
									wsNameId:= "off",
									wsName:= "off");	
	stText_GoTo		: ST_Text := (
									nNameId:= 1,
									wsNameId:= "goto",
									wsName:= "go to");	
									
	stText_JogPos		: ST_Text := (
									nNameId:= 1,
									wsNameId:= "jogpos",
									wsName:= "jog pos");

	stText_JogNeg		: ST_Text := (
									nNameId:= 1,
									wsNameId:= "jogneg",
									wsName:= "jog neg");
	
	stText_Gear			: ST_Text := (
									nNameId:= 1,
									wsNameId:= "gear",
									wsName:= "gear");
									
	stText_RefReset		: ST_Text :=  (
									nNameId:= 1,
									wsNameId:= "refreset",
									wsName:= "refreset");									
									
	stText_Brake		: ST_Text := (
									nNameId:= 1,
									wsNameId:= "brake",
									wsName:= "brake");	

	stText_SetPos		: ST_Text := (
									nNameId:= 1,
									wsNameId:= "setpos",
									wsName:= "setpos");								

	stText_Abspositioning		: ST_Text := (
									nNameId:= 1,
									wsNameId:= "abspositioning",
									wsName:= "abs positioning");
									
	stText_Jogpermanent		: ST_Text := (
									nNameId:= 1,
									wsNameId:= "jogpermanent",
									wsName:= "jog permanent");

	stText_Jog_0_001	: ST_Text := (
									nNameId:= 1,
									wsNameId:= "jog0_001",
									wsName:= "jog 0.001");

	stText_Jog_0_01	: ST_Text := (
									nNameId:= 1,
									wsNameId:= "jog0_01",
									wsName:= "jog 0.01");

	stText_Jog_0_1	: ST_Text := (
									nNameId:= 1,
									wsNameId:= "jog0_1",
									wsName:= "jog 0.1");

	stText_Jog_1_0	: ST_Text := (
									nNameId:= 1,
									wsNameId:= "jog1_0",
									wsName:= "jog 1.0");

	stText_Jog_10_0	: ST_Text := (
									nNameId:= 1,
									wsNameId:= "jog10_0",
									wsName:= "jog 10.0");
									
	stText_Mode_StartStop	: ST_Text := (
									nNameId:= 1,
									wsNameId:= "modestartstop",
									wsName:= "mode start stop");

	stText_Mode_Jog	: ST_Text := (
									nNameId:= 1,
									wsNameId:= "modejog",
									wsName:= "mode jog");									
											
	stText_Positive		: ST_Text := (
									nNameId:= 1,
									wsNameId:= "positive",
									wsName:= "positive");								

	stText_Negative		: ST_Text := (
									nNameId:= 1,
									wsNameId:= "negative",
									wsName:= "negative");	

	stText_Hp		: ST_Text := (
									nNameId:= 1,
									wsNameId:= "hp",
									wsName:= "hp");

	stText_Mp		: ST_Text := (
									nNameId:= 1,
									wsNameId:= "mp",
									wsName:= "mp");									

	stText_Wp		: ST_Text := (
									nNameId:= 1,
									wsNameId:= "wp",
									wsName:= "wp");	

	stText_emptymodeactive	: ST_Text := (
									nNameId:= 1,
									wsNameId:= "emptymodeactive",
									wsName:= "emptymodeactive");	

	stText_logout		: ST_Text := (
									nNameId:= 1,
									wsNameId:= "logout",
									wsName:= "logout");	
									
	stText_login		: ST_Text := (
									nNameId:= 1,
									wsNameId:= "login",
									wsName:= "login");	
									
	stText_submit		: ST_Text := (
									nNameId:= 1,
									wsNameId:= "submit",
									wsName:= "submit");
									
	stText_password		: ST_Text := (
									nNameId:= 1,
									wsNameId:= "password",
									wsName:= "password");	
									
	stText_UserLevel_None		: ST_Text := (
									nNameId:= 1,
									wsNameId:= "userlevelnone",
									wsName:= "none");

	stText_UserLevel_Programmer	: ST_Text := (
									nNameId:= 1,
									wsNameId:= "userlevelprogrammer",
									wsName:= "programmer");									
									
	stText_UserLevel_Admin	: ST_Text := (
									nNameId:= 1,
									wsNameId:= "userleveladmin",
									wsName:= "admin");	

	stText_UserLevel_Maintenance	: ST_Text := (
									nNameId:= 1,
									wsNameId:= "userlevelmaintenance",
									wsName:= "maintenance");	

	stText_UserLevel_Manager	: ST_Text := (
									nNameId:= 1,
									wsNameId:= "userlevelmanager",
									wsName:= "manager");	

	stText_UserLevel_Operator	: ST_Text := (
									nNameId:= 1,
									wsNameId:= "userleveloperator",
									wsName:= "operator");								
	//----------------------------------------------------------------------------------------------------
	//Notification Groups
	stText_NG_System				: ST_Text := (
									nNameId:= 1,
									wsNameId:= "System_Messages",
									wsName:= "System Messages");
									
	stText_NG_Hardware				: ST_Text := (
									nNameId:= 1,
									wsNameId:= "Hardware_Messages",
									wsName:= "Hardware Messages");
									
	stText_NG_Safety				: ST_Text := (
									nNameId:= 1,
									wsNameId:= "Safety_Notifications",
									wsName:= "Safety Notifications");
									
	stText_NG_Counter				: ST_Text := (
									nNameId:= 1,
									wsNameId:= "Counter_Notifications",
									wsName:= "Counter Notifications");									
									
									
	stText_NG_Modul001			: ST_Text := (
									nNameId:= 1,
									wsNameId:= "Modul001_Messages",
									wsName:= "Modul001 Messages");	

	stText_NG_Modul002			: ST_Text := (
									nNameId:= 1,
									wsNameId:= "Modul002_Messages",
									wsName:= "Modul002 Messages");

	stText_NG_Modul003			: ST_Text := (
									nNameId:= 1,
									wsNameId:= "Modul003_Messages",
									wsName:= "Modul003 Messages");

	stText_NG_Modul004			: ST_Text := (
									nNameId:= 1,
									wsNameId:= "Modul004_Messages",
									wsName:= "Modul004 Messages");								

	stText_NG_Stations				: ST_Text := (
									nNameId:= 1,
									wsNameId:= "Stations_Messages",
									wsName:= "Stations Messages");
									
	//----------------------------------------------------------------------------------------------------
	// Safety Messages
	stText_Safety					: ST_Text_List_Safety;
	//----------------------------------------------------------------------------------------------------
	//Order	
	stText_Order			: ST_Text := (
									nNameId:= 1,
									wsNameId:= "order",
									wsName:= "Auftrang");	
									
	stText_OrderNumber			: ST_Text := (
									nNameId:= 1,
									wsNameId:= "ordernumber",
									wsName:= "Auftrangsnummer");

	//----------------------------------------------------------------------------------------------------
	//Recipe
	stText_Recipe_Mode_None		: ST_Text := (
									nNameId:= 1,
									wsNameId:= "recipemode_none",
									wsName:= "kein Rezept");

	stText_Recipe_Mode_ToFrom	: ST_Text := (
									nNameId:= 1,
									wsNameId:= "recipemode_tofrom",
									wsName:= "Rezept <->");
							
	stText_000_Recipe			: ST_Text := (
									nNameId:= 1,
									wsNameId:= "000_recipe",
									wsName:= "000_recipe");										
									
	stText_Recipe				: ST_Text := (
									nNameId:= 1,
									wsNameId:= "[recipe]",
									wsName:= "[recipe]");	
	stText_RecipeName			: ST_Text := (
									nNameId:= 1,
									wsNameId:= "recipename",
									wsName:= "Recipename");									

	stText_RecipeComment		: ST_Text := (
									nNameId:= 1,
									wsNameId:= "RecipeComment",
									wsName:= "Comment");	

	stText_Recipe_SaveError		: ST_Text := (
									nNameId:= 1,
									wsNameId:= "Recipe_SaveError",
									wsName:= "Error saving recipe");	

	stText_Recipe_LoadError		: ST_Text := (
									nNameId:= 1,
									wsNameId:= "Recipe_LoadError",
									wsName:= "Error loading recipe");	

	stText_Recipe_ListError		: ST_Text := (
									nNameId:= 1,
									wsNameId:= "Recipe_ListError",
									wsName:= "Error list recipes");	

	stText_Recipe_CopyError		: ST_Text := (
									nNameId:= 1,
									wsNameId:= "Recipe_CopyError",
									wsName:= "Error copy recipe");	
									
	stText_Recipe_Loaded		: ST_Text := (
									nNameId:= 1,
									wsNameId:= "Recipe_Loaded",
									wsName:= "Recipe loaded");	
		
	//----------------------------------------------------------------------------------------------------
	//general	
	stText_None			: ST_Text := (
									nNameId:= 1,
									wsNameId:= "none",
									wsName:= "none");
						
	stText_Supervision			: ST_Text := (
									nNameId:= 1,
									wsNameId:= "Supervision",
									wsName:= "Supervision");

	stText_Info			: ST_Text := (
									nNameId:= 1,
									wsNameId:= "info",
									wsName:= "info");
			
	stText_Warning			: ST_Text := (
									nNameId:= 1,
									wsNameId:= "warning",
									wsName:= "warning");

	stText_Error			: ST_Text := (
									nNameId:= 1,
									wsNameId:= "error",
									wsName:= "error");						
						
	stText_Automatic		: ST_Text := (
									nNameId:= 1,
									wsNameId:= "automatic",
									wsName:= "automatic");	
									
	stText_Setup			: ST_Text := (
									nNameId:= 1,
									wsNameId:= "setup",
									wsName:= "setup");								
									
	stText_Auto				: ST_Text := (
									nNameId:= 1,
									wsNameId:= "auto",
									wsName:= "auto");

	stText_Manual			: ST_Text := (
									nNameId:= 1,
									wsNameId:= "manual",
									wsName:= "manual");

	stText_Step				: ST_Text := (
									nNameId:= 1,
									wsNameId:= "step",
									wsName:= "step");					

	stText_DeactivateModule	: ST_Text := (
									nNameId:= 1,
									wsNameId:= "deactivatemodule",
									wsName:= "deactivatemodule");
	
	stText_DeactivateStation	: ST_Text := (
									nNameId:= 1,
									wsNameId:= "deactivatestation",
									wsName:= "deactivatestation");

	stText_AutoHome				: ST_Text := (
									nNameId:= 1,
									wsNameId:= "autohome",
									wsName:= "auto home");	

	stText_PartReleaseInCaseOfHp	: ST_Text := (
									nNameId:= 1,
									wsNameId:= "partreleaseincaseofhp",
									wsName:= "part release in case of hp");									

	stText_CounterLimitNok		: ST_Text := (
									nNameId:= 1,
									wsNameId:= "counter limit nok",
									wsName:= "counter limit nok");	
									
	stText_Save					: ST_Text := (
									nNameId:= 1,
									wsNameId:= "save",
									wsName:= "save");
									
	stText_Autoreset				: ST_Text := (
									nNameId:= 1,
									wsNameId:= "autoreset",
									wsName:= "autoreset");
	
	stText_Userreset				: ST_Text := (
									nNameId:= 1,
									wsNameId:= "userreset",
									wsName:= "userreset");

	//----------------------------------------------------------------------------------------------------	
						
	//----------------------------------------------------------------------------------------------------
	
	stText_PlantName				: ST_Text := (
									nNameId:= 1,
									wsNameId:= "plantname",
									wsName:= "plant name");
	
	stText_PlantNumber				: ST_Text := (
									nNameId:= 1,
									wsNameId:= "plantnumber",
									wsName:= "plant number");

	stText_Plant_Absaugung_WachdogOn : ST_Text := (
									nNameId:= 1,
									wsNameId:= "anlageM3absaugungwachdogein",
									wsName:= "Anlage M3 Absaugung Wachdog ein");
								
	stText_Plant_Absaugung_WachdogOff : ST_Text := (
									nNameId:= 1,
									wsNameId:= "anlageM3absaugungwachdogaus",
									wsName:= "Anlage M3 Absaugung Wachdog aus");

	stText_Plant_Absaugung_Nachlauf : ST_Text := (
									nNameId:= 1,
									wsNameId:= "anlageM3absaugungnachlauf",
									wsName:= "Anlage M3 Absaugung Nachlauf");									
									

	stText_product		: ST_Text := (
									nNameId:= 1,
									wsNameId:= "product",
									wsName:= "product");
									
	stText_productnumber		: ST_Text := (
									nNameId:= 1,
									wsNameId:= "product_number",
									wsName:= "product number");

	stText_production	: ST_Text := (
									nNameId:= 1,
									wsNameId:= "production",
									wsName:= "production");
									
	stText_general			: ST_Text := (
									nNameId:= 1,
									wsNameId:= "general",
									wsName:= "general");	

	stText_Z_Reserve			: ST_Text := (
									nNameId:= 1,
									wsNameId:= "Z-Reserve",
									wsName:= "Z-Reserve");

	//----------------------------------------------------------------------------------------------------
	// HW Messages
	stText_EtherCatMaster_Error	: ST_Text := (
									nNameId:= 1,
									wsNameId:= "EtherCAT_Master_Error",
									wsName:= "EtherCAT Master Error");	

	stText_EtherCatBox_Error	: ST_Text := (
									nNameId:= 1,
									wsNameId:= "EtherCAT_Box_Error",
									wsName:= "EtherCAT Box Error");	
	stText_EtherCatBox_OP_Error	: ST_Text := (
									nNameId:= 1,
									wsNameId:= "EtherCAT_Box_OP_Error",
									wsName:= "EtherCAT Box OP-State Error");	

	stText_EtherCatSlave_Error	: ST_Text := (
									nNameId:= 1,
									wsNameId:= "EtherCAT_Slave_Error",
									wsName:= "EtherCAT Salve Error");	

	stText_Profinet_Error		: ST_Text := (
									nNameId:= 1,
									wsNameId:= "Profinet_Error",
									wsName:= "Profinet Error");	
									
	stText_NetGuard_Warn		: ST_Text := (
									nNameId:= 1,
									wsNameId:= "NetGuard_Error",
									wsName:= "NetGuard Error");	
	stText_NetGuard_Error		: ST_Text := (
									nNameId:= 1,
									wsNameId:= "NetGuard_Error",
									wsName:= "NetGuard Error");	

	stText_Cabinet_Warn			: ST_Text := (
									nNameId:= 1,
									wsNameId:= "Cabinet_Warn",
									wsName:= "Cabinet Warning");	
	stText_Cabinet_Error		: ST_Text := (
									nNameId:= 1,
									wsNameId:= "Cabinet_Error",
									wsName:= "Cabinet Error");	
	stText_Cabinet_Info		: ST_Text := (
									nNameId:= 1,
									wsNameId:= "Cabinet_Info",
									wsName:= "Cabinet Info");
							
	//----------------------------------------------------------------------------------------------------
	// Component messages
	stText_Comp					: ST_Text_List_Components;
	
	//----------------------------------------------------------------------------------------------------
	//generel plant
	stText_Drehwerkzeug			: ST_Text := (
									nNameId:= 1,
									wsNameId:= "drehwerkzeug",
									wsName:= "Drehwerkzeug");
	
	stText_Kontaktwerkzeug1	: ST_Text := (
									nNameId:= 1,
									wsNameId:= "kontaktwerkzeuglinks",
									wsName:= "Kontaktwerkzeug links");
									
	stText_Kontaktwerkzeug2		: ST_Text := (
									nNameId:= 1,
									wsNameId:= "kontaktwerkzeuglinks",
									wsName:= "Kontaktwerkzeug rechts");	

	stText_SchweisseinsatzAmboss		: ST_Text := (
									nNameId:= 1,
									wsNameId:= "schweisseinsatzAmboss",
									wsName:= "Schweisseinsatz Amboss");
	stText_SchweisseinsatzEinsatz		: ST_Text := (
									nNameId:= 1,
									wsNameId:= "schweisseinsatzEinsatz",
									wsName:= "Schweisseinsatz Einsatz");									

	stText_GreiferDatenReset	: ST_Text := (
									nNameId:= 1,
									wsNameId:= "GripperDataReset",
									wsName:= "Greifer Daten Löschen");
									
	stText_SetPosGs				: ST_Text := (
									nNameId:= 1,
									wsNameId:= "setposgs",
									wsName:= "Setze Position Gs");
									
	stText_SetPosMs				: ST_Text := (
									nNameId:= 1,
									wsNameId:= "setposms",
									wsName:= "Setze Position Ms");									

	stText_SetPosWt				: ST_Text := (
									nNameId:= 1,
									wsNameId:= "setposwt",
									wsName:= "Setze Position WT");

	stText_SetPosAusgabeIo		: ST_Text := (
									nNameId:= 1,
									wsNameId:= "setposausgabeio",
									wsName:= "Setze Position Ausgabe Io");	

	stText_SetPosAusgabeNio		: ST_Text := (
									nNameId:= 1,
									wsNameId:= "setposnioausgabenio",
									wsName:= "Setze Position Ausgabe Nio");								
	
	stText_BearbeitungStart: ST_Text := (
									nNameId:= 1,
									wsNameId:= "BearbeitungStart",
									wsName:= "Start Bearbeitung");
								
	stText_BearbeitungDatenReset: ST_Text := (
									nNameId:= 1,
									wsNameId:= "workingdatareset",
									wsName:= "Bearbeitung Daten Löschen");									

	stText_KameraProgramm: ST_Text := (
									nNameId:= 1,
									wsNameId:= "camprogram",
									wsName:= "Kamera Program");	
	stText_ProgrammLaden: ST_Text := (
									nNameId:= 1,
									wsNameId:= "ProgrammLaden",
									wsName:= "Programm Laden");	
									
	stText_KameraTrigger: ST_Text := (
									nNameId:= 1,
									wsNameId:= "camtrigger",
									wsName:= "Kamera Trigger");								

	//----------------------------------------------------------------------------------------------------
	//safety									
	stText_Emergencystop_A1P1	: ST_Text := (
									nNameId:= 1,
									wsNameId:= "emergencystopa1p1",
									wsName:= "Nothalt P1");	

	stText_Emergencystop_A1P2	: ST_Text := (
									nNameId:= 1,
									wsNameId:= "emergencystopa1p2",
									wsName:= "Nothalt P2");

	stText_Emergencystop_M1P1	: ST_Text := (
									nNameId:= 1,
									wsNameId:= "emergencystopm1p1",
									wsName:= "Nothalt M1 P1");
									
	stText_Emergencystop_M1P2	: ST_Text := (
									nNameId:= 1,
									wsNameId:= "emergencystopm1p2",
									wsName:= "Nothalt M1 P2");									

	stText_Emergencystop_M2P1	: ST_Text := (
									nNameId:= 1,
									wsNameId:= "emergencystopm2p1",
									wsName:= "Nothalt M2 P1");
									
	stText_Emergencystop_M3P1	: ST_Text := (
									nNameId:= 1,
									wsNameId:= "emergencystopm3p1",
									wsName:= "Nothalt M3 P1");	

	stText_Emergencystop_M3Laser1	: ST_Text := (
									nNameId:= 1,
									wsNameId:= "emergencystopm3laser1",
									wsName:= "Nothalt M3 Laser 1");	

	stText_Emergencystop_M3Laser2	: ST_Text := (
									nNameId:= 1,
									wsNameId:= "emergencystopm3laser2",
									wsName:= "Nothalt M3 Laser 2");

	stText_Emergencystop_M3Laser3	: ST_Text := (
									nNameId:= 1,
									wsNameId:= "emergencystopm3laser3",
									wsName:= "Nothalt M3 Laser 3");								

	stText_Emergencystop_M4P1	: ST_Text := (
									nNameId:= 1,
									wsNameId:= "emergencystopm4p1",
									wsName:= "Nothalt M4 P1");
									
	stText_Emergencystop_M4P2	: ST_Text := (
									nNameId:= 1,
									wsNameId:= "emergencystopm4p2",
									wsName:= "Nothalt M4 P2");							
	//----------------------------------------------------------------------------------------------------
	//modul
	stText_Modul1_Door1	: ST_Text := (
									nNameId:= 1,
									wsNameId:= "modul1door1",
									wsName:= "Modul 1 Tür 1");

	stText_Modul1_Door2	: ST_Text := (
									nNameId:= 1,
									wsNameId:= "modul1door2",
									wsName:= "Modul 1 Tür 2");

	stText_Modul1_Door3	: ST_Text := (
									nNameId:= 1,
									wsNameId:= "modul1door3",
									wsName:= "Modul 1 Tür 3");
									
	stText_Modul1_Door4	: ST_Text := (
									nNameId:= 1,
									wsNameId:= "modul1door4",
									wsName:= "Modul 1 Tür 4");								
									
	stText_Modul1_Schott1	: ST_Text := (
									nNameId:= 1,
									wsNameId:= "modul1schott1",
									wsName:= "Modul 1 Schott 1");	

	stText_Modul1_Schott2	: ST_Text := (
									nNameId:= 1,
									wsNameId:= "modul1schott2",
									wsName:= "Modul 1 Schott 2");								
							
	//----------------------------------------------------------------------------------------------------
	//stations
	
	stText_initialize_station	: ST_Text := (
									nNameId:= 1,
									wsNameId:= "initialize_station",
									wsName:= "initialize station");	
									
	stText_wait_for_start		: ST_Text := (
									nNameId:= 1,
									wsNameId:= "wait_for_start",
									wsName:= "wait for start");		

	stText_cycle_start			: ST_Text := (
									nNameId:= 1,
									wsNameId:= "cycle_start",
									wsName:= "cycle start");

	stText_wait_station_in_hp	: ST_Text := (
									nNameId:= 1,
									wsNameId:= "wait_station_in_hp",
									wsName:= "wait station in hp");	
								
	stText_station_not_in_hp	: ST_Text := (
									nNameId:= 1,
									wsNameId:= "station_not_in_hp",
									wsName:= "station not in hp");

	//-------------------------------------------
	//stations
	stText_M000_Name		: ST_Text := (
									nNameId:= 1,
									wsNameId:= "M000_Module",
									wsName:= "M000 Module");
									
	stText_M001_Name		: ST_Text := (
									nNameId:= 1,
									wsNameId:= "M001_Machine",
									wsName:= "M001 Machine");								
						
	
	//-------------------------------------------
	//stations
									
									

	//-------------------------------------------
	//stations 100
	stText_ST100_Name			: ST_Text := (
										nNameId:= 1,
										wsNameId:= "ST100_roundtable",
										wsName:= "ST100 Round Table");

	stText_ST100_NameId		: ST_Text := (
									nNameId:= 1,
									wsNameId:= "ST100",
									wsName:= "ST100");

	stText_ST100_Sequence	: ST_Text := (
									nNameId:= 1,
									wsNameId:= "tt",
									wsName:= "Rundtakttisch");
											

	stText_ST100_Axis			: ST_Text := (
										nNameId:= 1,
										wsNameId:= "ST100_Axis",
										wsName:= "Achsen St100");		
	stText_ST100_Drives			: ST_Text := (
										nNameId:= 1,
										wsNameId:= "ST100_Drives",
										wsName:= "Antriebe St100");		
	stText_ST100_Cyl			: ST_Text := (
										nNameId:= 1,
										wsNameId:= "ST100_Cyl",
										wsName:= "Zylinder St100");		
	stText_ST100_Sensor			: ST_Text := (
										nNameId:= 1,
										wsNameId:= "ST100_Sensor",
										wsName:= "Sensoren St100");
						
	stText_ST100_Setting_RttSpeedAuto			: ST_Text := (
										nNameId:= 1,
										wsNameId:= "ST100_SettingTtSpeedAuto",
										wsName:= "Setting St100 Speed Auto");
										
	stText_ST100_Setting_RttSpeedManual			: ST_Text := (
										nNameId:= 1,
										wsNameId:= "ST100_SettingTtSpeedManual",
										wsName:= "Setting St100 Speed Manual");	

	stText_ST100_TeileAmTransportsystem		: ST_Text := (
										nNameId:= 1,
										wsNameId:= "ST100TeileAmTransportsystem",
										wsName:= "ST100 Teile am Transportsystem");	

	stText_ST100_NioTeileAmTransportsystem		: ST_Text := (
										nNameId:= 1,
										wsNameId:= "ST100NioTeileAmTransportsystem",
										wsName:= "ST100 Nio Teile am Transportsystem");	

	stText_ST100_WorkstationActiveST001		: ST_Text := (
										nNameId:= 1,
										wsNameId:= "ST100WorkstationActiveST001",
										wsName:= "ST100 Workstation Active ST001");	

	stText_ST100_WorkstationActiveST002		: ST_Text := (
										nNameId:= 1,
										wsNameId:= "ST100WorkstationActiveST002",
										wsName:= "ST100 Workstation Active ST002");	

	stText_ST100_WorkstationActiveST003		: ST_Text := (
										nNameId:= 1,
										wsNameId:= "ST100WorkstationActiveST003",
										wsName:= "ST100 Workstation Active ST003");	

	stText_ST100_WorkstationActiveST004		: ST_Text := (
										nNameId:= 1,
										wsNameId:= "ST100WorkstationActiveST004",
										wsName:= "ST100 Workstation Active ST004");	

	stText_ST100_WorkstationActiveST005		: ST_Text := (
										nNameId:= 1,
										wsNameId:= "ST100WorkstationActiveST005",
										wsName:= "ST100 Workstation Active ST005");		

	stText_ST100_WorkstationPassableST001		: ST_Text := (
										nNameId:= 1,
										wsNameId:= "ST100WorkstationPassableST001",
										wsName:= "ST100 Workstation Passable ST001");	

	stText_ST100_WorkstationPassableST002		: ST_Text := (
										nNameId:= 1,
										wsNameId:= "ST100WorkstationPassableST002",
										wsName:= "ST100 Workstation Passable ST002");	

	stText_ST100_WorkstationPassableST003		: ST_Text := (
										nNameId:= 1,
										wsNameId:= "ST100WorkstationPassableST003",
										wsName:= "ST100 Workstation Passable ST003");	

	stText_ST100_WorkstationPassableST004		: ST_Text := (
										nNameId:= 1,
										wsNameId:= "ST100WorkstationPassableST004",
										wsName:= "ST100 Workstation Passable ST004");	

	stText_ST100_WorkstationPassableST005		: ST_Text := (
										nNameId:= 1,
										wsNameId:= "ST100WorkstationPassableST005",
										wsName:= "ST100 Workstation Passable ST005");	

	stText_ST100_WorkstationWorkEnableST001		: ST_Text := (
										nNameId:= 1,
										wsNameId:= "ST100WorkstationWorkEnableST001",
										wsName:= "ST100 Workstation WorkEnable ST001");	

	stText_ST100_WorkstationWorkEnableST002		: ST_Text := (
										nNameId:= 1,
										wsNameId:= "ST100WorkstationWorkEnableST002",
										wsName:= "ST100 Workstation WorkEnable ST002");	

	stText_ST100_WorkstationWorkEnableST003		: ST_Text := (
										nNameId:= 1,
										wsNameId:= "ST100WorkstationWorkEnableST003",
										wsName:= "ST100 Workstation WorkEnable ST003");	

	stText_ST100_WorkstationWorkEnableST004		: ST_Text := (
										nNameId:= 1,
										wsNameId:= "ST100WorkstationWorkEnableST004",
										wsName:= "ST100 Workstation WorkEnable ST004");	

	stText_ST100_WorkstationWorkEnableST005		: ST_Text := (
										nNameId:= 1,
										wsNameId:= "ST100WorkstationWorkEnableST005",
										wsName:= "ST100 Workstation WorkEnable ST005");	

	stText_ST100_WorkstationTurnEnableST001		: ST_Text := (
										nNameId:= 1,
										wsNameId:= "ST100WorkstationTurnEnableST001",
										wsName:= "ST100 Workstation TurnEnable ST001");	

	stText_ST100_WorkstationTurnEnableST002		: ST_Text := (
										nNameId:= 1,
										wsNameId:= "ST100WorkstationTurnEnableST002",
										wsName:= "ST100 Workstation TurnEnable ST002");	

	stText_ST100_WorkstationTurnEnableST003		: ST_Text := (
										nNameId:= 1,
										wsNameId:= "ST100WorkstationTurnEnableST003",
										wsName:= "ST100 Workstation TurnEnable ST003");	

	stText_ST100_WorkstationTurnEnableST004		: ST_Text := (
										nNameId:= 1,
										wsNameId:= "ST100WorkstationTurnEnableST004",
										wsName:= "ST100 Workstation TurnEnable ST004");	

	stText_ST100_WorkstationTurnEnableST005		: ST_Text := (
										nNameId:= 1,
										wsNameId:= "ST100WorkstationTurnEnableST005",
										wsName:= "ST100 Workstation TurnEnable ST005");		

	stText_ST100_Cycletime			: ST_Text := (
										nNameId:= 1,
										wsNameId:= "ST100Cycletime",
										wsName:= "ST100 Cycletime");	
			
	//----------------------------------------------------------------------------------------------------
	//axis
	stText_AxisXWp	: ST_Text := (
									nNameId:= 1,
									wsNameId:= "axis_x_wp",
									wsName:= "axis x wp");
									
	stText_AxisXHp	: ST_Text := (
									nNameId:= 1,
									wsNameId:= "axis_x_hp",
									wsName:= "axis x hp");								

	stText_AxisYWp	: ST_Text := (
									nNameId:= 1,
									wsNameId:= "axsis_y_wp",
									wsName:= "axis y wp");

	stText_AxisYHp	: ST_Text := (
									nNameId:= 1,
									wsNameId:= "axis_y_hp",
									wsName:= "axis y hp");									
									
	stText_AxisZWp	: ST_Text := (
									nNameId:= 1,
									wsNameId:= "limit_axsis_Z_wp",
									wsName:= "limit axsis Z wp");

	stText_AxisZHp	: ST_Text := (
									nNameId:= 1,
									wsNameId:= "axis_z_hp",
									wsName:= "axis z hp");

								
	//----------------------------------------------------------------------------------------------------
	//messages
	stText_AllOk	: ST_Text := (
									nNameId:= 1,
									wsNameId:= "allok",
									wsName:= "allok");
									
	stText_AxisZnotInHp	: ST_Text := (
									nNameId:= 1,
									wsNameId:= "axis_z_not_in_hp",
									wsName:= "axis z hp");

	//----------------------------------------------------------------------------------------------------
	//tc3hmi
	stText_Home		: ST_Text := (
									nNameId:= 1,
									wsNameId:= "home",
									wsName:= "home");	
	
	stText_Start	: ST_Text := (
									nNameId:= 1,
									wsNameId:= "start",
									wsName:= "start");
									
	stText_Stop		: ST_Text := (
									nNameId:= 1,
									wsNameId:= "stop",
									wsName:= "stop");
									
	stText_CycleStop: ST_Text := (
									nNameId:= 1,
									wsNameId:= "cyclestop",
									wsName:= "cyclestop");									
																		
	stText_Reset	: ST_Text := (
									nNameId:= 1,
									wsNameId:= "reset",
									wsName:= "reset");	
									
	stText_OPM_Auto	: ST_Text := (
									nNameId:= 1,
									wsNameId:= "opmauto",
									wsName:= "opmauto");									
									
	stText_OPM_Manual	: ST_Text := (
									nNameId:= 1,
									wsNameId:= "opmmanual",
									wsName:= "opmmanual");									

	stText_OPM_Step	: ST_Text := (
									nNameId:= 1,
									wsNameId:= "opmstep",
									wsName:= "opmstep");									

	stText_NavUser	: ST_Text := (
									nNameId:= 1,
									wsNameId:= "User",
									wsName:= "User");
	
	stText_PlantLight	: ST_Text := (
									nNameId:= 1,
									wsNameId:= "plantlight",
									wsName:= "Anlagenlicht");						
END_STRUCT
END_TYPE

// ---- POUs/HMI/_Structures/_TextLists/ST_Text_List_Safety.TcDUT
TYPE ST_Text_List_Safety :
STRUCT
	stText_Safety				: ST_Text := (
									wsNameId:= "Safety",
									wsName:= "Sicherheit");
									
	// Safety Messages
	stText_Safety_Grp_Error		: ST_Text := (
									wsNameId:= "Safety_group_Error",
									wsName:= "Fehler Safety-Gruppe");
	stText_Safety_GrpFB_Error	: ST_Text := (
									wsNameId:= "Safety_group_FB Error",
									wsName:= "Safety-Gruppe FB Fehler");
	stText_Safety_GrpCom_Error	: ST_Text := (
									wsNameId:= "Safety_group_Other_Error",
									wsName:= "Safety-Gruppe Fehler");
	stText_Safety_GrpOthError	: ST_Text := (
									wsNameId:= "Safety_group_COM_Error",
									wsName:= "Safety-Gruppe COM Fehler");
	stText_Safety_Error			: ST_Text := (
									wsNameId:= "Safety_Error",
									wsName:= "Safety Fehler");
	stText_Safety_ES			: ST_Text := (
									wsNameId:= "Emergency_stop",
									wsName:= "NOT-HALT");
	stText_Safety_Door			: ST_Text := (
									wsNameId:= "Safety_Door",
									wsName:= "Safety Tür");
	stText_Safety_DoorOpen		: ST_Text := (
									wsNameId:= "Safety_door_open",
									wsName:= "Safety Tür offen");
	stText_Safety_CloseDoor		: ST_Text := (
									wsNameId:= "Close_safety_door",
									wsName:= "Safety Tür schließen");
	stText_Safety_HW_Error		: ST_Text := (
									wsNameId:= "Safety_HW_Error",
									wsName:= "Safety Hardware Fehler");
	stText_Safety_FB_Error		: ST_Text := (
									wsNameId:= "Safety_FB_Error",
									wsName:= "Safety FB Fehler");
	stText_Safety_FB_Warning	: ST_Text := (
									wsNameId:= "Safety_FB_Warning",
									wsName:= "Safety FB Warnung");
	stText_Safety_EDM_Error		: ST_Text := (
									wsNameId:= "Safety_EDM_error",
									wsName:= "Safety EDM Fehler");
	stText_Safety_Discrepancy_Warning : ST_Text := (
									wsNameId:= "Safety_discrepancy_warning",
									wsName:= "Safety Diskrepanz Warnung (Button losgelassen)");
	stText_Safety_Discrepancy_Error : ST_Text := (
									wsNameId:= "Safety_discrepancy_error",
									wsName:= "Safety Diskrepanz Fehler");
	stText_Safety_2Hand_Error		: ST_Text := (
									wsNameId:= "Safety_2hand_error",
									wsName:= "Safety 2-Hand Fehler");
							
		
	stText_Safety_Error_Diagnosis : ST_Text := (
									wsNameId:= "Error_diagnosis",
									wsName:= "Fehler in Diagnose");
									
	stText_Safety_Error_SensortestInput : ST_Text := (
									wsNameId:= "Error_sensortest_input",
									wsName:= "Fehler Sensortest Eingang");
									
	stText_Safety_Error_FirstInputPair : ST_Text := (
									wsNameId:= "Error_first_input_pair",
									wsName:= "Fehler erstes Eingangspaar");
									
	stText_Safety_Error_SecondInputPair : ST_Text := (
									wsNameId:= "Error_second_input_pair",
									wsName:= "Fehler zweites Eingangspaar");
									
	stText_Safety_Error_ExternalSupplyOutput : ST_Text := (
									wsNameId:= "Error_external_supply_output",
									wsName:= "Fehler externe Versorgung Ausgang");
									
	stText_Safety_Error_OpenLoadOutput : ST_Text := (
									wsNameId:= "Error_OpenLoad_output",
									wsName:= "Fehler keine Last am Ausgang");
									
	stText_Safety_Error_FieldVoltageToHigh : ST_Text := (
									wsNameId:= "Error_field_voltage_to_high",
									wsName:= "Fehler Feldspannung zu hoch");
									
	stText_Safety_Error_FieldVoltageToLow : ST_Text := (
									wsNameId:= "Error_field_voltage_to_low",
									wsName:= "Fehler Feldspannung zu niedrig");
									
									
	stText_Safety_Error_Temperature : ST_Text := (
									wsNameId:= "Error_temperature",
									wsName:= "Fehler Temperatur");
									
	stText_Safety_Error_OutputTerminal : ST_Text := (
									wsNameId:= "Error_output_terminal",
									wsName:= "Fehler Ausgangs-Terminal");
									
									
	stText_Safety_TimerSwitchOnTimeout	: ST_Text := (
									wsNameId:= "Safety_Timer_Switch_On_Timeout",
									wsName:= "Timer 'Switch On' Timeout");
								
	stText_Safety_TimerSwitchOffTimeout	: ST_Text := (
									wsNameId:= "Safety_Timer_Switch_Off_Timeout",
									wsName:= "Timer 'Switch Off' Timeout");
END_STRUCT
END_TYPE

// ---- POUs/HMI/_Structures/_TextLists/ST_Text_List_System.TcDUT
TYPE ST_Text_List_System :
STRUCT
	stText_CycletimeExceeded				: ST_Text := (
												wsNameId:= "CycletimeExceeded",
												wsName:= "Zykluszeit Überschreitung");
												
	stText_CodeError					: ST_Text := (
												wsNameId:= "CodeError",
												wsName:= "Code Fehler");

	// EtherCAT master
	stText_EC_CommonError					: ST_Text := (
												wsNameId:= "EC_CommonError",
												wsName:= "Allg. EtherCAT Fehler");
	stText_EC_LinkError						: ST_Text := (
												wsNameId:= "EC_LinkError",
												wsName:= "Link error");
	stText_EC_IoLockedAfterLinkErr			: ST_Text := (
												wsNameId:= "EC_IoLockedAfterLinkErr",
												wsName:= "I/O locked after link error (I/O reset required)");
	stText_EC_LinkErrRedAdapter				: ST_Text := (
												wsNameId:= "EC_LinkErrRedAdapter",
												wsName:= "Link error (redundancy adapter)");
	stText_EC_MissingFrame					: ST_Text := (
												wsNameId:= "EC_MissingFrame",
												wsName:= "Missing one frame (redundancy mode)");
	stText_EC_OutOfSendResources			: ST_Text := (
												wsNameId:= "EC_OutOfSendResources",
												wsName:= "Out of send resources (I/O reset required)");												
	stText_EC_WatchdogTriggered				: ST_Text := (
												wsNameId:= "EC_WatchdogTriggered",
												wsName:= "Watchdog triggered");												
	stText_EC_EthernetDrvNotFound			: ST_Text := (
												wsNameId:= "EC_EthernetDrvNotFound",
												wsName:= "Ethernet driver (miniport) not found");												
	stText_EC_IO_resetActive				: ST_Text := (
												wsNameId:= "EC_IO_resetActive",
												wsName:= "I/O reset active");
	stText_EC_AtLeastOneDeviceInit			: ST_Text := (
												wsNameId:= "EC_AtLeastOneDeviceInit",
												wsName:= "At least one device in INIT state");
	stText_EC_AtLeastOneDevicePreOp			: ST_Text := (
												wsNameId:= "EC_AtLeastOneDevicePreOp",
												wsName:= "At least one device in PRE-OP state");
	stText_EC_AtLeastOneDeviceSafeOp		: ST_Text := (
												wsNameId:= "EC_AtLeastOneDeviceSafeOp",
												wsName:= "At least one device in SAFE-OP state");
	stText_EC_AtLeastOneDeviceError			: ST_Text := (
												wsNameId:= "EC_AtLeastOneDeviceError",
												wsName:= "At least one device indicates an error state");
	stText_EC_DC_notInSync					: ST_Text := (
												wsNameId:= "EC_DC_notInSync",
												wsName:= "DC not in sync");
	stText_SystemStartupReset				: ST_Text := (
												wsNameId:= "SystemReStart_Reset",
												wsName:= "System (re)start, press reset.");
												
